(* Logix 5000 project; controller VET 1756-L62 rev 19.52; software revision 19.01; part 4 of 27 *)

        [24].S.BITS1.4   // 7-RED-1024 Cmd. Automatico
        [24].S.BITS1.29   // 90-CAN-011 Falla Abrir
        [24].S.BITS2.20   // 7-RED-1024 Reset Falla
        [24].S.BITS2.23   // 7-RED-1024 Test
        [24].S.BITS2.31   // 90-CAN-011 OUT OPEN
        [28].S.BITS1.0   // 90-VEN-006 Enable
        [28].S.BITS1.1   // 90-VEN-006 Falla Resumen
        [28].S.BITS1.2   // 90-VEN-006 Conf. Marcha
        [28].S.BITS1.4   // 90-VEN-006 Cmd. Automatico
        [28].S.BITS1.26   // 90-VEN-006 FLL
        [28].S.BITS1.27   // 90-VEN-006 FV0
        [28].S.BITS1.28   // 90-VEN-006 FATO
        [28].S.BITS1.30   // 90-VEN-006 Falla Partida
        [28].S.BITS2.27   // 90-VEN-006 Cmd. Marcha
        [28].S.BITS2.20   // 90-VEN-006 Reset Falla
        [28].S.BITS2.23   // 90-VEN-006 Test
        [28].S.BITS2.30   // 90-VEN-006 OUT MARCHA
        [29].S.BITS1.0   // 7-RED-1050 Enable
        [29].S.BITS1.1   // 7-RED-1050 Falla Resumen
        [29].S.BITS1.2   // 7-RED-1050 Conf. Marcha
        [29].S.BITS1.4   // 7-RED-1050 Cmd. Automatico
        [29].S.BITS1.26   // 7-RED-1050 FLL
        [29].S.BITS1.27   // 7-RED-1050 FV0
        [29].S.BITS1.28   // 7-RED-1050 FATO
        [29].S.BITS1.30   // 7-RED-1050 Falla Partida
        [29].S.BITS2.27   // 7-RED-1050 Cmd. Marcha
        [29].S.BITS2.20   // 7-RED-1050 Reset Falla
        [29].S.BITS2.23   // 7-RED-1050 Test
        [29].S.BITS2.30   // 7-RED-1050 OUT MARCHA
        [31].S.BITS1.8   // 90-TOL-001 LL
        [31].S.BITS1.9   // 90-TOL-001 LM
        [31].S.BITS1.10   // 90-TOL-001 LH
        [33].S.BITS1.10   // 90-TOL-003 LH
        [33].S.BITS1.8   // 90-TOL-003 LL
        [33].S.BITS1.9   // 90-TOL-003 LM
        [35].S.BITS1.8   // 90-TOL-005 LL
        [34].S.BITS1.8   // 90-TOL-004 LL
        [37].S.BITS1.10   // 90-TOL-007 LH
        [36].S.BITS1.8   // 7-BIN-1060 LL
        [37].S.BITS1.8   // 90-TOL-007 LL
        [37].S.BITS1.9   // 90-TOL-007 LM
        [40].S.BITS2.30   // 7-VRT-1064 OUT MARCHA
        [43].S.BITS2.30   // 7-VEN-1067 OUT MARCHA
        [44].S.BITS1.2   // 90-FIL-001 Conf Pos Abrir
        [44].S.BITS1.29   // 90-FIL-001 Falla Abrir
        [44].S.BITS2.31   // 90-FIL-001 OUT OPEN
        [45].S.BITS1.26   // 7-ROS-1068 FLL
        [45].S.BITS1.27   // 7-ROS-1068 FV0
        [45].S.BITS1.28   // 7-ROS-1068 FATO
        [45].S.BITS1.30   // 7-ROS-1068 Falla Partida
        [45].S.BITS2.27   // 7-ROS-1068 Cmd. Marcha
        [45].S.BITS2.30   // 7-ROS-1068 OUT MARCHA
        [47].S.BITS1.8   // TV-1 LL
        [47].S.BITS1.10   // TV-1 LH
        [55].S.BITS1.2   // 7-RED-1078 Conf. Marcha
        [55].S.BITS1.29   // 90-FIL-002 Falla Abrir
        [55].S.BITS2.31   // 90-FIL-002 OUT OPEN
        [56].S.BITS1.26   // 90-VEN-002 FLL
        [56].S.BITS1.27   // 90-VEN-002 FV0
        [56].S.BITS1.28   // 90-VEN-002 FATO
        [56].S.BITS1.30   // 7-CON-1079 Falla Cerrar
        [56].S.BITS2.27   // 7-CON-1079 Cmd. Open
        [56].S.BITS2.30   // 7-CON-1079 OUT CLOSE
        [59].S.BITS1.27   // 90-TOR-002 FV0
        [58].S.BITS1.8   // TV-2 LL
        [59].S.BITS1.0   // 90-TOR-002 Enable
        [59].S.BITS1.1   // 90-TOR-002 Falla Resumen
        [59].S.BITS1.2   // 90-TOR-002 Conf. Marcha
        [59].S.BITS1.4   // 90-TOR-002 Cmd. Automatico
        [59].S.BITS1.26   // 90-TOR-002 FLL
        [59].S.BITS1.28   // 90-TOR-002 FATO
        [59].S.BITS1.30   // 90-TOR-002 Falla Partida
        [59].S.BITS2.27   // 90-TOR-002 Cmd. Marcha
        [59].S.BITS2.20   // 90-TOR-002 Reset Falla
        [59].S.BITS2.23   // 90-TOR-002 Test
        [59].S.BITS2.30   // 90-TOR-002 OUT MARCHA
        [63].S.BITS1.0   // 7-MRO-1083c Enable
        [63].S.BITS1.1   // 7-MRO-1083c Falla Resumen
        [63].S.BITS1.2   // 7-MRO-1083c Conf. Marcha
        [63].S.BITS1.4   // 7-MRO-1083c Cmd. Automatico
        [63].S.BITS1.26   // 7-MRO-1083c FLL
        [63].S.BITS1.27   // 7-MRO-1083c FV0
        [63].S.BITS1.28   // 7-MRO-1083c FATO
        [63].S.BITS1.30   // 7-MRO-1083c Falla Partida
        [63].S.BITS2.27   // 7-MRO-1083c Cmd. Marcha
        [63].S.BITS2.20   // 7-MRO-1083c Reset Falla
        [63].S.BITS2.23   // 7-MRO-1083c Test
        [63].S.BITS2.30   // 7-MRO-1083c OUT MARCHA
        [64].S.BITS1.0   // 7-MRO-1083d Enable
        [64].S.BITS1.1   // 7-MRO-1083d Falla Resumen
        [64].S.BITS1.2   // 7-MRO-1083d Conf. Marcha
        [64].S.BITS1.4   // 7-MRO-1083d Cmd. Automatico
        [64].S.BITS1.26   // 7-MRO-1083d FLL
        [64].S.BITS1.27   // 7-MRO-1083d FV0
        [64].S.BITS1.28   // 7-MRO-1083d FATO
        [64].S.BITS1.30   // 7-MRO-1083d Falla Partida
        [64].S.BITS2.27   // 7-MRO-1083d Cmd. Marcha
        [64].S.BITS2.20   // 7-MRO-1083d Reset Falla
        [64].S.BITS2.23   // 7-MRO-1083d Test
        [64].S.BITS2.30   // 7-MRO-1083d OUT MARCHA
        [65].S.BITS1.0   // 90-MRO-001-C Enable
        [65].S.BITS1.1   // 90-MRO-001-C Falla Resumen
        [65].S.BITS1.2   // 90-MRO-001-C Conf. Marcha
        [65].S.BITS1.4   // 90-MRO-001-C Cmd. Automatico
        [65].S.BITS1.26   // 90-MRO-001-C FLL
        [65].S.BITS1.27   // 90-MRO-001-C FV0
        [65].S.BITS1.28   // 90-MRO-001-C FATO
        [65].S.BITS1.30   // 90-MRO-001-C Falla Partida
        [65].S.BITS2.27   // 90-MRO-001-C Cmd. Marcha
        [65].S.BITS2.20   // 90-MRO-001-C Reset Falla
        [65].S.BITS2.23   // 90-MRO-001-C Test
        [65].S.BITS2.30   // 90-MRO-001-C OUT MARCHA
        [72].S.BITS1.2   // 90-ALI-004 Conf. Marcha
        [73].S.BITS1.0   // 7-MRO-1089a Enable
        [73].S.BITS1.1   // 7-MRO-1089a Falla Resumen
        [73].S.BITS1.2   // 7-MRO-1089a Conf. Marcha
        [73].S.BITS1.4   // 7-MRO-1089a Cmd. Automatico
        [73].S.BITS1.26   // 7-MRO-1089a FLL
        [73].S.BITS1.27   // 7-MRO-1089a FV0
        [73].S.BITS1.28   // 7-MRO-1089a FATO
        [73].S.BITS1.30   // 7-MRO-1089a Falla Partida
        [73].S.BITS2.27   // 7-MRO-1089a Cmd. Marcha
        [73].S.BITS2.20   // 7-MRO-1089a Reset Falla
        [73].S.BITS2.23   // 7-MRO-1089a Test
        [73].S.BITS2.30   // 7-MRO-1089a OUT MARCHA
        [74].S.BITS1.0   // 7-MRO-1089b Enable
        [74].S.BITS1.1   // 7-MRO-1089b Falla Resumen
        [74].S.BITS1.4   // 7-MRO-1089b Cmd. Automatico
        [74].S.BITS1.26   // 7-MRO-1089b FLL
        [74].S.BITS1.27   // 7-MRO-1089b FV0
        [74].S.BITS1.28   // 7-MRO-1089b FATO
        [74].S.BITS1.30   // 7-MRO-1089b Falla Partida
        [74].S.BITS2.27   // 7-MRO-1089b Cmd. Marcha
        [74].S.BITS2.20   // 7-MRO-1089b Reset Falla
        [74].S.BITS2.23   // 7-MRO-1089b Test
        [74].S.BITS2.30   // 7-MRO-1089b OUT MARCHA
        [75].S.BITS1.0   // 7-MRO-1089c Enable
        [75].S.BITS1.1   // 7-MRO-1089c Falla Resumen
        [75].S.BITS1.2   // 7-MRO-1089c Conf. Marcha
        [75].S.BITS1.4   // 7-MRO-1089c Cmd. Automatico
        [75].S.BITS1.26   // 7-MRO-1089c FLL
        [75].S.BITS1.27   // 7-MRO-1089c FV0
        [75].S.BITS1.28   // 7-MRO-1089c FATO
        [75].S.BITS1.30   // 7-MRO-1089c Falla Partida
        [75].S.BITS2.27   // 7-MRO-1089c Cmd. Marcha
        [75].S.BITS2.20   // 7-MRO-1089c Reset Falla
        [75].S.BITS2.23   // 7-MRO-1089c Test
        [75].S.BITS2.30   // 7-MRO-1089c OUT MARCHA
        [82].S.BITS1.0   // 7-CON-1095 Enable
        [82].S.BITS1.1   // 7-CON-1095 Falla Resumen
        [82].S.BITS1.4   // 7-CON-1095 Conf Pos Cerrar
        [82].S.BITS1.26   // 90-ALI-005 FLL
        [82].S.BITS1.27   // 90-ALI-005 FV0
        [82].S.BITS1.28   // 90-ALI-005 FATO
        [82].S.BITS1.30   // 7-CON-1095 Falla Cerrar
        [82].S.BITS2.27   // 7-CON-1095 Cmd. Open
        [82].S.BITS2.20   // 7-CON-1095 Reset Falla
        [82].S.BITS2.23   // 7-CON-1095 Test
        [82].S.BITS2.30   // 7-CON-1095 OUT CLOSE
        [83].S.BITS1.0   // 7-CON-1096 Enable
        [83].S.BITS1.1   // 7-CON-1096 Falla Resumen
        [83].S.BITS1.2   // 7-CON-1096 Conf Pos Abrir
        [83].S.BITS1.4   // 7-CON-1096 Conf Pos Cerrar
        [83].S.BITS1.26   // 90-MRO-003-A FLL
        [83].S.BITS1.27   // 90-MRO-003-A FV0
        [83].S.BITS1.28   // 90-MRO-003-A FATO
        [83].S.BITS1.30   // 7-CON-1096 Falla Cerrar
        [83].S.BITS2.27   // 7-CON-1096 Cmd. Open
        [83].S.BITS2.20   // 7-CON-1096 Reset Falla
        [83].S.BITS2.23   // 7-CON-1096 Test
        [83].S.BITS2.30   // 7-CON-1096 OUT CLOSE
        [84].S.BITS1.0   // 7-CON-1097 Enable
        [84].S.BITS1.1   // 7-CON-1097 Falla Resumen
        [84].S.BITS1.4   // 7-CON-1097 Conf Pos Cerrar
        [84].S.BITS1.26   // 90-MRO-003-B FLL
        [84].S.BITS1.27   // 90-MRO-003-B FV0
        [84].S.BITS1.28   // 90-MRO-003-B FATO
        [84].S.BITS1.30   // 7-CON-1097 Falla Cerrar
        [84].S.BITS2.27   // 7-CON-1097 Cmd. Open
        [84].S.BITS2.20   // 7-CON-1097 Reset Falla
        [84].S.BITS2.23   // 7-CON-1097 Test
        [84].S.BITS2.30   // 7-CON-1097 OUT CLOSE
        [85].S.BITS1.0   // 90-MRO-003-C Enable
        [85].S.BITS1.1   // 90-MRO-003-C Falla Resumen
        [85].S.BITS1.4   // 90-MRO-003-C Cmd. Automatico
        [85].S.BITS1.26   // 90-MRO-003-C FLL
        [85].S.BITS1.27   // 90-MRO-003-C FV0
        [85].S.BITS1.28   // 90-MRO-003-C FATO
        [85].S.BITS1.30   // 90-MRO-003-C Falla Partida
        [85].S.BITS2.27   // 90-MRO-003-C Cmd. Marcha
        [85].S.BITS2.20   // 90-MRO-003-C Reset Falla
        [85].S.BITS2.23   // 90-MRO-003-C Test
        [85].S.BITS2.30   // 90-MRO-003-C OUT MARCHA
        [92].S.BITS1.0   // 90-VEN-003 Enable
        [92].S.BITS1.1   // 90-VEN-003 Falla Resumen
        [92].S.BITS1.2   // 90-VEN-003 Conf. Marcha
        [92].S.BITS1.4   // 90-VEN-003 Cmd. Automatico
        [92].S.BITS1.26   // 90-VEN-003 FLL
        [92].S.BITS1.27   // 90-VEN-003 FV0
        [92].S.BITS1.28   // 90-VEN-003 FATO
        [92].S.BITS1.30   // 90-VEN-003 Falla Partida
        [92].S.BITS2.27   // 90-VEN-003 Cmd. Marcha
        [92].S.BITS2.20   // 90-VEN-003 Reset Falla
        [92].S.BITS2.23   // 90-VEN-003 Test
        [92].S.BITS2.30   // 90-VEN-003 OUT MARCHA
        [96].S.BITS1.27   // 90-TDC-006 FV0
        [94].S.BITS1.8   // 90-TOL-008 LL
        [94].S.BITS1.9   // 90-TOL-008 LM
        [94].S.BITS1.10   // 90-TOL-008 LH
        [96].S.BITS1.0   // 90-TDC-006 Enable
        [96].S.BITS1.1   // 90-TDC-006 Falla Resumen
        [96].S.BITS1.4   // 90-TDC-006 Cmd. Automatico
        [96].S.BITS1.26   // 90-TDC-006 FLL
        [96].S.BITS1.28   // 90-TDC-006 FATO
        [96].S.BITS1.30   // 90-TDC-006 Falla Partida
        [96].S.BITS2.27   // 90-TDC-006 Cmd. Marcha
        [96].S.BITS2.20   // 90-TDC-006 Reset Falla
        [96].S.BITS2.23   // 90-TDC-006 Test
        [96].S.BITS2.30   // 90-TDC-006 OUT MARCHA
        [97].S.BITS1.0   // 90-CAN-019 Enable
        [97].S.BITS1.1   // 90-CAN-019 Falla Resumen
        [97].S.BITS1.2   // 90-CAN-019 Conf Pos Abrir
        [97].S.BITS1.4   // 90-CAN-019 Conf Pos Cerrar
        [97].S.BITS1.29   // 90-CAN-019 Falla Abrir
        [97].S.BITS1.30   // 90-CAN-019 Falla Cerrar
        [97].S.BITS2.20   // 90-CAN-019 Reset Falla
        [97].S.BITS2.23   // 90-CAN-019 Test
        [97].S.BITS2.27   // 90-CAN-019 Cmd. Open
        [97].S.BITS2.30   // 90-CAN-019 OUT CLOSE
        [97].S.BITS2.31   // 90-CAN-019 OUT OPEN
        [101].S.BITS1.8   // 7-BIN-1100 LL
        [99].S.BITS1.9   // TOLVIR-MRO1 LM
        [102].S.BITS1.1   // 7-ROS-1101 Falla Resumen
        [100].S.BITS1.8   // TOLVIR-MRO2 LL
        [100].S.BITS1.9   // TOLVIR-MRO2 LM
        [100].S.BITS1.10   // TOLVIR-MRO2 LH
        [102].S.BITS1.27   // 7-ROS-1101 FV0
        [101].S.BITS1.9   // 7-BIN-1100 LM
        [101].S.BITS1.10   // 7-BIN-1100 LH
        [102].S.BITS1.0   // 7-ROS-1101 Enable
        [102].S.BITS1.2   // 7-ROS-1101 Conf. Marcha
        [102].S.BITS1.4   // 7-ROS-1101 Cmd. Automatico
        [102].S.BITS1.26   // 7-ROS-1101 FLL
        [102].S.BITS1.28   // 7-ROS-1101 FATO
        [102].S.BITS1.30   // 7-ROS-1101 Falla Partida
        [102].S.BITS2.27   // 7-ROS-1101 Cmd. Marcha
        [102].S.BITS2.20   // 7-ROS-1101 Reset Falla
        [102].S.BITS2.23   // 7-ROS-1101 Test
        [102].S.BITS2.30   // 7-ROS-1101 OUT MARCHA
        [104].S.BITS1.0   // 7-ROS-1103 Enable
        [104].S.BITS1.1   // 7-ROS-1103 Falla Resumen
        [104].S.BITS1.2   // 7-ROS-1103 Conf. Marcha
        [104].S.BITS1.4   // 7-ROS-1103 Cmd. Automatico
        [104].S.BITS1.26   // 7-ROS-1103 FLL
        [104].S.BITS1.27   // 7-ROS-1103 FV0
        [104].S.BITS1.28   // 7-ROS-1103 FATO
        [104].S.BITS1.30   // 7-ROS-1103 Falla Partida
        [104].S.BITS2.27   // 7-ROS-1103 Cmd. Marcha
        [104].S.BITS2.20   // 7-ROS-1103 Reset Falla
        [104].S.BITS2.23   // 7-ROS-1103 Test
        [104].S.BITS2.30   // 7-ROS-1103 OUT MARCHA
        [105].S.BITS1.0   // 90-TDC-004 Enable
        [105].S.BITS1.1   // 90-TDC-004 Falla Resumen
        [105].S.BITS1.2   // 90-TDC-004 Conf. Marcha
        [105].S.BITS1.4   // 90-TDC-004 Cmd. Automatico
        [105].S.BITS1.26   // 90-TDC-004 FLL
        [105].S.BITS1.27   // 90-TDC-004 FV0
        [105].S.BITS1.28   // 90-TDC-004 FATO
        [105].S.BITS1.30   // 90-TDC-004 Falla Partida
        [105].S.BITS2.27   // 90-TDC-004 Cmd. Marcha
        [105].S.BITS2.20   // 90-TDC-004 Reset Falla
        [105].S.BITS2.23   // 90-TDC-004 Test
        [105].S.BITS2.30   // 90-TDC-004 OUT MARCHA
        [106].S.BITS1.0   // 7-ROS-1105 Enable
        [106].S.BITS1.1   // 7-ROS-1105 Falla Resumen
        [106].S.BITS1.4   // 7-ROS-1105 Cmd. Automatico
        [106].S.BITS1.26   // 7-ROS-1105 FLL
        [106].S.BITS1.27   // 7-ROS-1105 FV0
        [106].S.BITS1.28   // 7-ROS-1105 FATO
        [106].S.BITS1.30   // 7-ROS-1105 Falla Partida
        [106].S.BITS2.27   // 7-ROS-1105 Cmd. Marcha
        [106].S.BITS2.20   // 7-ROS-1105 Reset Falla
        [106].S.BITS2.23   // 7-ROS-1105 Test
        [106].S.BITS2.30   // 7-ROS-1105 OUT MARCHA
        [107].S.BITS1.0   // 90-ELV-002 Enable
        [107].S.BITS1.1   // 90-ELV-002 Falla Resumen
        [107].S.BITS1.2   // 90-ELV-002 Conf. Marcha
        [107].S.BITS1.4   // 90-ELV-002 Cmd. Automatico
        [107].S.BITS1.26   // 90-ELV-002 FLL
        [107].S.BITS1.27   // 90-ELV-002 FV0
        [107].S.BITS1.28   // 90-ELV-002 FATO
        [107].S.BITS1.30   // 90-ELV-002 Falla Partida
        [107].S.BITS2.27   // 90-ELV-002 Cmd. Marcha
        [107].S.BITS2.20   // 90-ELV-002 Reset Falla
        [107].S.BITS2.23   // 90-ELV-002 Test
        [107].S.BITS2.30   // 90-ELV-002 OUT MARCHA
        [109].S.BITS1.0   // 90-ELV-004 Enable
        [109].S.BITS1.1   // 90-ELV-004 Falla Resumen
        [109].S.BITS1.4   // 90-ELV-004 Cmd. Automatico
        [109].S.BITS1.26   // 90-ELV-004 FLL
        [109].S.BITS1.27   // 90-ELV-004 FV0
        [109].S.BITS1.28   // 90-ELV-004 FATO
        [109].S.BITS1.30   // 90-ELV-004 Falla Partida
        [109].S.BITS2.27   // 90-ELV-004 Cmd. Marcha
        [109].S.BITS2.20   // 90-ELV-004 Reset Falla
        [109].S.BITS2.23   // 90-ELV-004 Test
        [109].S.BITS2.30   // 90-ELV-004 OUT MARCHA
        [112].S.BITS1.0   // 7-ROS-1111 Enable
        [112].S.BITS1.1   // 7-ROS-1111 Falla Resumen
        [112].S.BITS1.2   // 7-ROS-1111 Conf. Marcha
        [112].S.BITS1.4   // 7-ROS-1111 Cmd. Automatico
        [112].S.BITS1.26   // 7-ROS-1111 FLL
        [112].S.BITS1.27   // 7-ROS-1111 FV0
        [112].S.BITS1.28   // 7-ROS-1111 FATO
        [112].S.BITS1.30   // 7-ROS-1111 Falla Partida
        [112].S.BITS2.27   // 7-ROS-1111 Cmd. Marcha
        [112].S.BITS2.20   // 7-ROS-1111 Reset Falla
        [112].S.BITS2.23   // 7-ROS-1111 Test
        [112].S.BITS2.30   // 7-ROS-1111 OUT MARCHA
        [113].S.BITS1.0   // 100-VEN-001 Enable
        [113].S.BITS1.1   // 100-VEN-001 Falla Resumen
        [113].S.BITS1.2   // 100-VEN-001 Conf. Marcha
        [113].S.BITS1.4   // 100-VEN-001 Cmd. Automatico
        [113].S.BITS1.26   // 100-VEN-001 FLL
        [113].S.BITS1.27   // 100-VEN-001 FV0
        [113].S.BITS1.28   // 100-VEN-001 FATO
        [113].S.BITS1.30   // 100-VEN-001 Falla Partida
        [113].S.BITS2.27   // 100-VEN-001 Cmd. Marcha
        [113].S.BITS2.20   // 100-VEN-001 Reset Falla
        [113].S.BITS2.23   // 100-VEN-001 Test
        [113].S.BITS2.30   // 100-VEN-001 OUT MARCHA
        [115].S.BITS1.27   // 100-TOR-022 FV0
        [114].S.BITS1.8   // 100-TOL-005 LL
        [114].S.BITS1.9   // 100-TOL-005 LM
        [114].S.BITS1.10   // 100-TOL-005 LH
        [115].S.BITS1.0   // 100-TOR-022 Enable
        [115].S.BITS1.1   // 100-TOR-022 Falla Resumen
        [115].S.BITS1.4   // 100-TOR-022 Cmd. Automatico
        [115].S.BITS1.26   // 100-TOR-022 FLL
        [115].S.BITS1.28   // 100-TOR-022 FATO
        [115].S.BITS1.30   // 100-TOR-022 Falla Partida
        [115].S.BITS2.27   // 100-TOR-022 Cmd. Marcha
        [115].S.BITS2.20   // 100-TOR-022 Reset Falla
        [115].S.BITS2.23   // 100-TOR-022 Test
        [115].S.BITS2.30   // 100-TOR-022 OUT MARCHA
        [116].S.BITS1.0   // 7-ROS-1115 Enable
        [116].S.BITS1.1   // 7-ROS-1115 Falla Resumen
        [116].S.BITS1.4   // 7-ROS-1115 Cmd. Automatico
        [116].S.BITS1.26   // 7-ROS-1115 FLL
        [116].S.BITS1.27   // 7-ROS-1115 FV0
        [116].S.BITS1.28   // 7-ROS-1115 FATO
        [116].S.BITS1.30   // 7-ROS-1115 Falla Partida
        [116].S.BITS2.27   // 7-ROS-1115 Cmd. Marcha
        [116].S.BITS2.20   // 7-ROS-1115 Reset Falla
        [116].S.BITS2.23   // 7-ROS-1115 Test
        [116].S.BITS2.30   // 7-ROS-1115 OUT MARCHA
        [117].S.BITS1.0   // 100-BIF-001 Enable
        [117].S.BITS1.1   // 100-BIF-001 Falla Resumen
        [117].S.BITS1.2   // 100-BIF-001 Conf. Pos. Izquierda
        [117].S.BITS1.4   // 100-BIF-001 Conf. Pos. Derecha
        [117].S.BITS1.29   // 100-BIF-001 Falla Pos. Izquierda
        [117].S.BITS1.30   // 100-BIF-001 Falla Pos. Derecha
        [117].S.BITS2.20   // 100-BIF-001 Reset Falla
        [117].S.BITS2.23   // 100-BIF-001 Test
        [117].S.BITS2.26   // 100-BIF-001 Cmd. Pos . Izquierda
        [117].S.BITS2.27   // 100-BIF-001 Cmd. Pos. Derecha
        [117].S.BITS2.30   // 100-BIF-001 Out Izquierda
        [117].S.BITS2.31   // 100-BIF-001 Out Derecha
        [122].S.BITS1.0   // 7-ROS-1121 Enable
        [122].S.BITS1.1   // 7-ROS-1121 Falla Resumen
        [122].S.BITS1.2   // 7-ROS-1121 Conf. Marcha
        [122].S.BITS1.4   // 7-ROS-1121 Cmd. Automatico
        [122].S.BITS1.26   // 7-ROS-1121 FLL
        [122].S.BITS1.27   // 7-ROS-1121 FV0
        [122].S.BITS1.28   // 7-ROS-1121 FATO
        [122].S.BITS1.30   // 7-ROS-1121 Falla Partida
        [122].S.BITS2.27   // 7-ROS-1121 Cmd. Marcha
        [122].S.BITS2.20   // 7-ROS-1121 Reset Falla
        [122].S.BITS2.23   // 7-ROS-1121 Test
        [122].S.BITS2.30   // 7-ROS-1121 OUT MARCHA
        [123].S.BITS1.0   // 100-CAN-018 Enable
        [123].S.BITS1.1   // 100-CAN-018 Falla Resumen
        [123].S.BITS1.2   // 100-CAN-018 Conf Pos Abrir
        [123].S.BITS1.4   // 100-CAN-018 Conf Pos Cerrar
        [123].S.BITS1.29   // 100-CAN-018 Falla Abrir
        [123].S.BITS2.20   // 100-CAN-018 Reset Falla
        [123].S.BITS2.23   // 100-CAN-018 Test
        [123].S.BITS2.31   // 100-CAN-018 OUT OPEN
        [124].S.BITS1.0   // 7-ROS-1123 Enable
        [124].S.BITS1.1   // 7-ROS-1123 Falla Resumen
        [124].S.BITS1.2   // 7-ROS-1123 Conf. Marcha
        [124].S.BITS1.4   // 7-ROS-1123 Cmd. Automatico
        [124].S.BITS1.29   // 100-CAN-019 Falla Abrir
        [124].S.BITS1.30   // 7-ROS-1123 Falla Partida
        [124].S.BITS2.20   // 7-ROS-1123 Reset Falla
        [124].S.BITS2.23   // 7-ROS-1123 Test
        [124].S.BITS2.30   // 7-ROS-1123 OUT MARCHA
        [124].S.BITS2.31   // 100-CAN-019 OUT OPEN
        [126].S.BITS1.0   // 7-ROS-1125 Enable
        [126].S.BITS1.1   // 7-ROS-1125 Falla Resumen
        [126].S.BITS1.2   // 7-ROS-1125 Conf. Marcha
        [126].S.BITS1.4   // 7-ROS-1125 Cmd. Automatico
        [126].S.BITS1.26   // 7-ROS-1125 FLL
        [126].S.BITS1.27   // 7-ROS-1125 FV0
        [126].S.BITS1.28   // 7-ROS-1125 FATO
        [126].S.BITS1.30   // 7-ROS-1125 Falla Partida
        [126].S.BITS2.27   // 7-ROS-1125 Cmd. Marcha
        [126].S.BITS2.20   // 7-ROS-1125 Reset Falla
        [126].S.BITS2.23   // 7-ROS-1125 Test
        [126].S.BITS2.30   // 7-ROS-1125 OUT MARCHA
        [127].S.BITS1.0   // 100-CAN-020 Enable
        [127].S.BITS1.1   // 100-CAN-020 Falla Resumen
        [127].S.BITS1.2   // 100-CAN-020 Conf Pos Abrir
        [127].S.BITS1.4   // 100-CAN-020 Conf Pos Cerrar
        [127].S.BITS1.29   // 100-CAN-020 Falla Abrir
        [127].S.BITS2.20   // 100-CAN-020 Reset Falla
        [127].S.BITS2.23   // 100-CAN-020 Test
        [127].S.BITS2.31   // 100-CAN-020 OUT OPEN
        [128].S.BITS1.0   // 7-ROS-1127 Enable
        [128].S.BITS1.1   // 7-ROS-1127 Falla Resumen
        [128].S.BITS1.2   // 7-ROS-1127 Conf. Marcha
        [128].S.BITS1.4   // 7-ROS-1127 Cmd. Automatico
        [128].S.BITS1.29   // 100-CAN-021 Falla Abrir
        [128].S.BITS1.30   // 7-ROS-1127 Falla Partida
        [128].S.BITS2.20   // 7-ROS-1127 Reset Falla
        [128].S.BITS2.23   // 7-ROS-1127 Test
        [128].S.BITS2.30   // 7-ROS-1127 OUT MARCHA
        [128].S.BITS2.31   // 100-CAN-021 OUT OPEN
        [131].S.BITS1.0   // 100-TDC-001 Enable
        [131].S.BITS1.1   // 100-TDC-001 Falla Resumen
        [131].S.BITS1.4   // 100-TDC-001 Cmd. Automatico
        [131].S.BITS1.26   // 100-TDC-001 FLL
        [131].S.BITS1.27   // 100-TDC-001 FV0
        [131].S.BITS1.28   // 100-TDC-001 FATO
        [131].S.BITS1.30   // 100-TDC-001 Falla Partida
        [131].S.BITS2.27   // 100-TDC-001 Cmd. Marcha
        [131].S.BITS2.20   // 100-TDC-001 Reset Falla
        [131].S.BITS2.23   // 100-TDC-001 Test
        [131].S.BITS2.30   // 100-TDC-001 OUT MARCHA
        [132].S.BITS1.0   // 100-CAN-001 Enable
        [132].S.BITS1.1   // 100-CAN-001 Falla Resumen
        [132].S.BITS1.2   // 100-CAN-001 Conf Pos Abrir
        [132].S.BITS1.4   // 100-CAN-001 Conf Pos Cerrar
        [132].S.BITS1.29   // 100-CAN-001 Falla Abrir
        [132].S.BITS1.30   // 100-CAN-001 Falla Cerrar
        [132].S.BITS2.20   // 100-CAN-001 Reset Falla
        [132].S.BITS2.23   // 100-CAN-001 Test
        [132].S.BITS2.27   // 100-CAN-001 Cmd. Open
        [132].S.BITS2.30   // 100-CAN-001 OUT CLOSE
        [132].S.BITS2.31   // 100-CAN-001 OUT OPEN
        [134].S.BITS1.0   // 100-TDC-002 Enable
        [134].S.BITS1.1   // 100-TDC-002 Falla Resumen
        [134].S.BITS1.2   // 100-TDC-002 Conf. Marcha
        [134].S.BITS1.4   // 100-TDC-002 Cmd. Automatico
        [134].S.BITS1.26   // 100-TDC-002 FLL
        [134].S.BITS1.27   // 100-TDC-002 FV0
        [134].S.BITS1.28   // 100-TDC-002 FATO
        [134].S.BITS1.30   // 100-TDC-002 Falla Partida
        [134].S.BITS2.27   // 100-TDC-002 Cmd. Marcha
        [134].S.BITS2.20   // 100-TDC-002 Reset Falla
        [134].S.BITS2.23   // 100-TDC-002 Test
        [134].S.BITS2.30   // 100-TDC-002 OUT MARCHA
        [135].S.BITS1.0   // 100-CAN-002 Enable
        [135].S.BITS1.1   // 100-CAN-002 Falla Resumen
        [135].S.BITS1.2   // 100-CAN-002 Conf Pos Abrir
        [135].S.BITS1.4   // 100-CAN-002 Conf Pos Cerrar
        [135].S.BITS1.29   // 100-CAN-002 Falla Abrir
        [135].S.BITS1.30   // 100-CAN-002 Falla Cerrar
        [135].S.BITS2.20   // 100-CAN-002 Reset Falla
        [135].S.BITS2.23   // 100-CAN-002 Test
        [135].S.BITS2.27   // 100-CAN-002 Cmd. Open
        [135].S.BITS2.30   // 100-CAN-002 OUT CLOSE
        [135].S.BITS2.31   // 100-CAN-002 OUT OPEN
        [136].S.BITS1.0   // 100-CAN-003 Enable
        [136].S.BITS1.1   // 100-CAN-003 Falla Resumen
        [136].S.BITS1.2   // 100-CAN-003 Conf Pos Abrir
        [136].S.BITS1.4   // 100-CAN-003 Conf Pos Cerrar
        [136].S.BITS1.29   // 100-CAN-003 Falla Abrir
        [136].S.BITS1.30   // 100-CAN-003 Falla Cerrar
        [136].S.BITS2.20   // 100-CAN-003 Reset Falla
        [136].S.BITS2.23   // 100-CAN-003 Test
        [136].S.BITS2.27   // 100-CAN-003 Cmd. Open
        [136].S.BITS2.30   // 100-CAN-003 OUT CLOSE
        [137].S.BITS1.0   // 100-CAN-004 Enable
        [137].S.BITS1.1   // 100-CAN-004 Falla Resumen
        [137].S.BITS1.2   // 100-CAN-004 Conf Pos Abrir
        [137].S.BITS1.4   // 100-CAN-004 Conf Pos Cerrar
        [137].S.BITS1.29   // 100-CAN-004 Falla Abrir
        [137].S.BITS1.30   // 100-CAN-004 Falla Cerrar
        [137].S.BITS2.20   // 100-CAN-004 Reset Falla
        [137].S.BITS2.23   // 100-CAN-004 Test
        [137].S.BITS2.27   // 100-CAN-004 Cmd. Open
        [137].S.BITS2.30   // 100-CAN-004 OUT CLOSE
        [137].S.BITS2.31   // 100-CAN-004 OUT OPEN
        [142].S.BITS1.0   // 7-FIL-1141 Enable
        [142].S.BITS1.1   // 7-FIL-1141 Falla Resumen
        [142].S.BITS1.2   // 7-FIL-1141 Conf. Marcha
        [142].S.BITS1.4   // 7-FIL-1141 Cmd. Automatico
        [142].S.BITS1.26   // 7-FIL-1141 FLL
        [142].S.BITS1.27   // 7-FIL-1141 FV0
        [142].S.BITS1.28   // 7-FIL-1141 FATO
        [142].S.BITS1.30   // 7-FIL-1141 Falla Partida
        [142].S.BITS2.27   // 7-FIL-1141 Cmd. Marcha
        [142].S.BITS2.20   // 7-FIL-1141 Reset Falla
        [142].S.BITS2.23   // 7-FIL-1141 Test
        [142].S.BITS2.30   // 7-FIL-1141 OUT MARCHA
        [143].S.BITS1.0   // 7-BBA-1142 Enable
        [143].S.BITS1.1   // 7-BBA-1142 Falla Resumen
        [143].S.BITS1.2   // 7-BBA-1142 Conf. Marcha
        [143].S.BITS1.4   // 7-BBA-1142 Cmd. Automatico
        [143].S.BITS1.29   // 100-CAN-005 Falla Abrir
        [143].S.BITS2.20   // 7-BBA-1142 Reset Falla
        [143].S.BITS2.23   // 7-BBA-1142 Test
        [143].S.BITS2.31   // 100-CAN-005 OUT OPEN
        [144].S.BITS1.0   // 7-RED-1143 Enable
        [144].S.BITS1.1   // 7-RED-1143 Falla Resumen
        [144].S.BITS1.2   // 7-RED-1143 Conf. Marcha
        [144].S.BITS1.4   // 7-RED-1143 Cmd. Automatico
        [144].S.BITS1.29   // 100-CAN-006 Falla Abrir
        [144].S.BITS1.30   // 7-RED-1143 Falla Partida
        [144].S.BITS2.20   // 7-RED-1143 Reset Falla
        [144].S.BITS2.23   // 7-RED-1143 Test
        [144].S.BITS2.30   // 7-RED-1143 OUT MARCHA
        [144].S.BITS2.31   // 100-CAN-006 OUT OPEN
        [146].S.BITS1.0   // 7-RED-1145 Enable
        [146].S.BITS1.1   // 7-RED-1145 Falla Resumen
        [146].S.BITS1.2   // 7-RED-1145 Conf. Marcha
        [146].S.BITS1.4   // 7-RED-1145 Cmd. Automatico
        [146].S.BITS1.26   // 7-RED-1145 FLL
        [146].S.BITS1.27   // 7-RED-1145 FV0
        [146].S.BITS1.28   // 7-RED-1145 FATO
        [146].S.BITS1.30   // 7-RED-1145 Falla Partida
        [146].S.BITS2.27   // 7-RED-1145 Cmd. Marcha
        [146].S.BITS2.20   // 7-RED-1145 Reset Falla
        [146].S.BITS2.23   // 7-RED-1145 Test
        [146].S.BITS2.30   // 7-RED-1145 OUT MARCHA
        [147].S.BITS1.0   // 7-CON-1146 Enable
        [147].S.BITS1.1   // 7-CON-1146 Falla Resumen
        [147].S.BITS1.2   // 7-CON-1146 Conf Pos Abrir
        [147].S.BITS1.4   // 7-CON-1146 Conf Pos Cerrar
        [147].S.BITS1.29   // 7-CON-1146 Falla Abrir
        [147].S.BITS2.20   // 7-CON-1146 Reset Falla
        [147].S.BITS2.23   // 7-CON-1146 Test
        [147].S.BITS2.31   // 7-CON-1146 OUT OPEN
        [148].S.BITS1.0   // 7-CON-1147 Enable
        [148].S.BITS1.1   // 7-CON-1147 Falla Resumen
        [148].S.BITS1.2   // 7-CON-1147 Conf Pos Abrir
        [148].S.BITS1.4   // 7-CON-1147 Conf Pos Cerrar
        [148].S.BITS1.29   // 7-CON-1147 Falla Abrir
        [148].S.BITS1.30   // 7-CON-1147 Falla Cerrar
        [148].S.BITS2.20   // 7-CON-1147 Reset Falla
        [148].S.BITS2.23   // 7-CON-1147 Test
        [148].S.BITS2.27   // 7-CON-1147 Cmd. Open
        [148].S.BITS2.30   // 7-CON-1147 OUT CLOSE
        [148].S.BITS2.31   // 7-CON-1147 OUT OPEN
        [152].S.BITS1.0   // 7-CON-1152 Enable
        [152].S.BITS1.1   // 7-CON-1152 Falla Resumen
        [152].S.BITS1.4   // 7-CON-1152 Conf Pos Cerrar
        [152].S.BITS1.26   // 100-TDC-005 FLL
        [152].S.BITS1.27   // 100-TDC-005 FV0
        [152].S.BITS1.28   // 100-TDC-005 FATO
        [152].S.BITS1.30   // 7-CON-1152 Falla Cerrar
        [152].S.BITS2.27   // 7-CON-1152 Cmd. Open
        [152].S.BITS2.20   // 7-CON-1152 Reset Falla
        [152].S.BITS2.23   // 7-CON-1152 Test
        [152].S.BITS2.30   // 7-CON-1152 OUT CLOSE
        [153].S.BITS1.0   // 7-CON-1153 Enable
        [153].S.BITS1.1   // 7-CON-1153 Falla Resumen
        [153].S.BITS1.2   // 7-CON-1153 Conf Pos Abrir
        [153].S.BITS1.4   // 7-CON-1153 Conf Pos Cerrar
        [153].S.BITS1.29   // 7-CON-1153 Falla Abrir
        [153].S.BITS2.20   // 7-CON-1153 Reset Falla
        [153].S.BITS2.23   // 7-CON-1153 Test
        [153].S.BITS2.31   // 7-CON-1153 OUT OPEN
        [154].S.BITS1.0   // 7-ELV-1149 Enable
        [154].S.BITS1.1   // 7-ELV-1149 Falla Resumen
        [154].S.BITS1.2   // 7-ELV-1149 Conf. Marcha
        [154].S.BITS1.4   // 7-ELV-1149 Cmd. Automatico
        [154].S.BITS1.29   // 100-CAN-014 Falla Abrir
        [154].S.BITS1.30   // 7-ELV-1149 Falla Partida
        [154].S.BITS2.20   // 7-ELV-1149 Reset Falla
        [154].S.BITS2.23   // 7-ELV-1149 Test
        [154].S.BITS2.30   // 7-ELV-1149 OUT MARCHA
        [154].S.BITS2.31   // 100-CAN-014 OUT OPEN
        [155].S.BITS1.0   // 100-CAN-015 Enable
        [155].S.BITS1.1   // 100-CAN-015 Falla Resumen
        [155].S.BITS1.2   // 100-CAN-015 Conf Pos Abrir
        [155].S.BITS1.4   // 100-CAN-015 Conf Pos Cerrar
        [155].S.BITS1.29   // 100-CAN-015 Falla Abrir
        [155].S.BITS2.20   // 100-CAN-015 Reset Falla
        [155].S.BITS2.23   // 100-CAN-015 Test
        [155].S.BITS2.31   // 100-CAN-015 OUT OPEN
        [157].S.BITS1.0   // 7-ROS-1156 Enable
        [157].S.BITS1.1   // 7-ROS-1156 Falla Resumen
        [157].S.BITS1.2   // 7-ROS-1156 Conf. Marcha
        [157].S.BITS1.4   // 7-ROS-1156 Cmd. Automatico
        [157].S.BITS1.26   // 7-ROS-1156 FLL
        [157].S.BITS1.27   // 7-ROS-1156 FV0
        [157].S.BITS1.28   // 7-ROS-1156 FATO
        [157].S.BITS1.30   // 7-ROS-1156 Falla Partida
        [157].S.BITS2.27   // 7-ROS-1156 Cmd. Marcha
        [157].S.BITS2.20   // 7-ROS-1156 Reset Falla
        [157].S.BITS2.23   // 7-ROS-1156 Test
        [157].S.BITS2.30   // 7-ROS-1156 OUT MARCHA
        [158].S.BITS1.0   // 100-CAN-016 Enable
        [158].S.BITS1.1   // 100-CAN-016 Falla Resumen
        [158].S.BITS1.2   // 100-CAN-016 Conf Pos Abrir
        [158].S.BITS1.4   // 100-CAN-016 Conf Pos Cerrar
        [158].S.BITS1.29   // 100-CAN-016 Falla Abrir
        [158].S.BITS1.30   // 100-CAN-016 Falla Cerrar
        [158].S.BITS2.20   // 100-CAN-016 Reset Falla
        [158].S.BITS2.23   // 100-CAN-016 Test
        [158].S.BITS2.27   // 100-CAN-016 Cmd. Open
        [158].S.BITS2.30   // 100-CAN-016 OUT CLOSE
        [158].S.BITS2.31   // 100-CAN-016 OUT OPEN
        [159].S.BITS1.0   // 7-ROS-1158 Enable
        [159].S.BITS1.1   // 7-ROS-1158 Falla Resumen
        [159].S.BITS1.2   // 7-ROS-1158 Conf. Marcha
        [159].S.BITS1.4   // 7-ROS-1158 Cmd. Automatico
        [159].S.BITS1.29   // 100-CAN-017 Falla Abrir
        [159].S.BITS2.20   // 7-ROS-1158 Reset Falla
        [159].S.BITS2.23   // 7-ROS-1158 Test
        [159].S.BITS2.31   // 100-CAN-017 OUT OPEN
        [162].S.BITS1.0   // 100-TDC-008 Enable
        [162].S.BITS1.1   // 100-TDC-008 Falla Resumen
        [162].S.BITS1.2   // 100-TDC-008 Conf. Marcha
        [162].S.BITS1.4   // 100-TDC-008 Cmd. Automatico
        [162].S.BITS1.26   // 100-TDC-008 FLL
        [162].S.BITS1.27   // 100-TDC-008 FV0
        [162].S.BITS1.28   // 100-TDC-008 FATO
        [162].S.BITS1.30   // 100-TDC-008 Falla Partida
        [162].S.BITS2.27   // 100-TDC-008 Cmd. Marcha
        [162].S.BITS2.20   // 100-TDC-008 Reset Falla
        [162].S.BITS2.23   // 100-TDC-008 Test
        [162].S.BITS2.30   // 100-TDC-008 OUT MARCHA
        [163].S.BITS1.0   // 7-ROS-1162 Enable
        [163].S.BITS1.1   // 7-ROS-1162 Falla Resumen
        [163].S.BITS1.2   // 7-ROS-1162 Conf. Marcha
        [163].S.BITS1.4   // 7-ROS-1162 Cmd. Automatico
        [163].S.BITS1.29   // 100-CAN-028 Falla Abrir
        [163].S.BITS2.20   // 7-ROS-1162 Reset Falla
        [163].S.BITS2.23   // 7-ROS-1162 Test
        [163].S.BITS2.31   // 100-CAN-028 OUT OPEN
        [164].S.BITS1.0   // 100-BIF-002 Enable
        [164].S.BITS1.1   // 100-BIF-002 Falla Resumen
        [164].S.BITS1.2   // 100-BIF-002 Conf. Pos. Izquierda
        [164].S.BITS1.4   // 100-BIF-002 Conf. Pos. Derecha
        [164].S.BITS1.29   // 100-BIF-002 Falla Pos. Izquierda
        [164].S.BITS1.30   // 100-BIF-002 Falla Pos. Derecha
        [164].S.BITS2.20   // 100-BIF-002 Reset Falla
        [164].S.BITS2.23   // 100-BIF-002 Test
        [164].S.BITS2.26   // 100-BIF-002 Cmd. Pos . Izquierda
        [164].S.BITS2.27   // 100-BIF-002 Cmd. Pos. Derecha
        [164].S.BITS2.30   // 100-BIF-002 Out Izquierda
        [164].S.BITS2.31   // 100-BIF-002 Out Derecha
        [165].S.BITS1.0   // 7-ROS-1164 Enable
        [165].S.BITS1.1   // 7-ROS-1164 Falla Resumen
        [165].S.BITS1.2   // 7-ROS-1164 Conf. Marcha
        [165].S.BITS1.4   // 7-ROS-1164 Cmd. Automatico
        [165].S.BITS1.29   // 100-BIF-003 Falla Pos. Izquierda
        [165].S.BITS1.30   // 7-ROS-1164 Falla Partida
        [165].S.BITS2.20   // 7-ROS-1164 Reset Falla
        [165].S.BITS2.23   // 7-ROS-1164 Test
        [165].S.BITS2.26   // 100-BIF-003 Cmd. Pos . Izquierda
        [165].S.BITS2.27   // 7-ROS-1164 Cmd. Marcha
        [165].S.BITS2.30   // 7-ROS-1164 OUT MARCHA
        [165].S.BITS2.31   // 100-BIF-003 Out Derecha
        [167].S.BITS1.0   // 7-ROS-1166 Enable
        [167].S.BITS1.1   // 7-ROS-1166 Falla Resumen
        [167].S.BITS1.2   // 7-ROS-1166 Conf. Marcha
        [167].S.BITS1.4   // 7-ROS-1166 Cmd. Automatico
        [167].S.BITS1.26   // 7-ROS-1166 FLL
        [167].S.BITS1.27   // 7-ROS-1166 FV0
        [167].S.BITS1.28   // 7-ROS-1166 FATO
        [167].S.BITS1.30   // 7-ROS-1166 Falla Partida
        [167].S.BITS2.27   // 7-ROS-1166 Cmd. Marcha
        [167].S.BITS2.20   // 7-ROS-1166 Reset Falla
        [167].S.BITS2.23   // 7-ROS-1166 Test
        [167].S.BITS2.30   // 7-ROS-1166 OUT MARCHA
        [168].S.BITS1.0   // 100-FIL-002 Enable
        [168].S.BITS1.1   // 100-FIL-002 Falla Resumen
        [168].S.BITS1.2   // 100-FIL-002 Conf. Marcha
        [168].S.BITS1.4   // 100-FIL-002 Cmd. Automatico
        [168].S.BITS1.26   // 100-FIL-002 FLL
        [168].S.BITS1.27   // 100-FIL-002 FV0
        [168].S.BITS1.28   // 100-FIL-002 FATO
        [168].S.BITS1.30   // 100-FIL-002 Falla Partida
        [168].S.BITS2.27   // 100-FIL-002 Cmd. Marcha
        [168].S.BITS2.20   // 100-FIL-002 Reset Falla
        [168].S.BITS2.23   // 100-FIL-002 Test
        [168].S.BITS2.30   // 100-FIL-002 OUT MARCHA
        [169].S.BITS1.0   // 100-VEN-002 Enable
        [169].S.BITS1.1   // 100-VEN-002 Falla Resumen
        [169].S.BITS1.2   // 100-VEN-002 Conf. Marcha
        [169].S.BITS1.4   // 100-VEN-002 Cmd. Automatico
        [169].S.BITS1.26   // 100-VEN-002 FLL
        [169].S.BITS1.27   // 100-VEN-002 FV0
        [169].S.BITS1.28   // 100-VEN-002 FATO
        [169].S.BITS1.30   // 100-VEN-002 Falla Partida
        [169].S.BITS2.27   // 100-VEN-002 Cmd. Marcha
        [169].S.BITS2.20   // 100-VEN-002 Reset Falla
        [169].S.BITS2.23   // 100-VEN-002 Test
        [169].S.BITS2.30   // 100-VEN-002 OUT MARCHA
        [172].S.BITS1.27   // 100-TOR-001 FV0
        [171].S.BITS1.8   // 100-BIN-001 LL
        [171].S.BITS1.9   // 100-BIN-001 LM
        [171].S.BITS1.10   // 100-BIN-001 LH
        [172].S.BITS1.0   // 100-TOR-001 Enable
        [172].S.BITS1.1   // 100-TOR-001 Falla Resumen
        [172].S.BITS1.2   // 100-TOR-001 Conf. Marcha
        [172].S.BITS1.4   // 100-TOR-001 Cmd. Automatico
        [172].S.BITS1.26   // 100-TOR-001 FLL
        [172].S.BITS1.28   // 100-TOR-001 FATO
        [172].S.BITS1.30   // 100-TOR-001 Falla Partida
        [172].S.BITS2.27   // 100-TOR-001 Cmd. Marcha
        [172].S.BITS2.20   // 100-TOR-001 Reset Falla
        [172].S.BITS2.23   // 100-TOR-001 Test
        [172].S.BITS2.30   // 100-TOR-001 OUT MARCHA
        [178].S.BITS1.27   // 100-TOR-003 FV0
        [177].S.BITS1.8   // 100-BIN-003 LL
        [177].S.BITS1.9   // 100-BIN-003 LM
        [177].S.BITS1.10   // 100-BIN-003 LH
        [178].S.BITS1.0   // 100-TOR-003 Enable
        [178].S.BITS1.1   // 100-TOR-003 Falla Resumen
        [178].S.BITS1.2   // 100-TOR-003 Conf. Marcha
        [178].S.BITS1.4   // 100-TOR-003 Cmd. Automatico
        [178].S.BITS1.26   // 100-TOR-003 FLL
        [178].S.BITS1.28   // 100-TOR-003 FATO
        [178].S.BITS1.30   // 100-TOR-003 Falla Partida
        [178].S.BITS2.27   // 100-TOR-003 Cmd. Marcha
        [178].S.BITS2.20   // 100-TOR-003 Reset Falla
        [178].S.BITS2.23   // 100-TOR-003 Test
        [178].S.BITS2.30   // 100-TOR-003 OUT MARCHA
        [182].S.BITS1.0   // 100-TOR-037 Enable
        [182].S.BITS1.1   // 100-TOR-037 Falla Resumen
        [182].S.BITS1.2   // 100-TOR-037 Conf. Marcha
        [182].S.BITS1.4   // 100-TOR-037 Cmd. Automatico
        [182].S.BITS1.26   // 100-TOR-037 FLL
        [182].S.BITS1.27   // 100-TOR-037 FV0
        [182].S.BITS1.28   // 100-TOR-037 FATO
        [182].S.BITS1.30   // 100-TOR-037 Falla Partida
        [182].S.BITS2.27   // 100-TOR-037 Cmd. Marcha
        [182].S.BITS2.20   // 100-TOR-037 Reset Falla
        [182].S.BITS2.23   // 100-TOR-037 Test
        [182].S.BITS2.30   // 100-TOR-037 OUT MARCHA
        [184].S.BITS1.27   // 100-TOR-005 FV0
        [183].S.BITS1.8   // 100-BIN-005 LL
        [183].S.BITS1.9   // 100-BIN-005 LM
        [183].S.BITS1.10   // 100-BIN-005 LH
        [184].S.BITS1.0   // 100-TOR-005 Enable
        [184].S.BITS1.1   // 100-TOR-005 Falla Resumen
        [184].S.BITS1.2   // 100-TOR-005 Conf. Marcha
        [184].S.BITS1.4   // 100-TOR-005 Cmd. Automatico
        [184].S.BITS1.26   // 100-TOR-005 FLL
        [184].S.BITS1.28   // 100-TOR-005 FATO
        [184].S.BITS1.30   // 100-TOR-005 Falla Partida
        [184].S.BITS2.27   // 100-TOR-005 Cmd. Marcha
        [184].S.BITS2.20   // 100-TOR-005 Reset Falla
        [184].S.BITS2.23   // 100-TOR-005 Test
        [184].S.BITS2.30   // 100-TOR-005 OUT MARCHA
        [196].S.BITS1.27   // 100-TOR-008 FV0
        [195].S.BITS1.9   // 100-BIN-008 LM
        [196].S.BITS1.0   // 100-TOR-008 Enable
        [196].S.BITS1.1   // 100-TOR-008 Falla Resumen
        [196].S.BITS1.2   // 100-TOR-008 Conf. Marcha
        [196].S.BITS1.4   // 100-TOR-008 Cmd. Automatico
        [196].S.BITS1.26   // 100-TOR-008 FLL
        [196].S.BITS1.28   // 100-TOR-008 FATO
        [196].S.BITS1.30   // 100-TOR-008 Falla Partida
        [196].S.BITS2.27   // 100-TOR-008 Cmd. Marcha
        [196].S.BITS2.20   // 100-TOR-008 Reset Falla
        [196].S.BITS2.23   // 100-TOR-008 Test
        [196].S.BITS2.30   // 100-TOR-008 OUT MARCHA
        [199].S.BITS1.27   // 100-TOR-009 FV0
        [198].S.BITS1.8   // 100-BIN-009 LL
        [198].S.BITS1.9   // 100-BIN-009 LM
        [198].S.BITS1.10   // 100-BIN-009 LH
        [199].S.BITS1.0   // 100-TOR-009 Enable
        [199].S.BITS1.1   // 100-TOR-009 Falla Resumen
        [199].S.BITS1.2   // 100-TOR-009 Conf. Marcha
        [199].S.BITS1.4   // 100-TOR-009 Cmd. Automatico
        [199].S.BITS1.26   // 100-TOR-009 FLL
        [199].S.BITS1.28   // 100-TOR-009 FATO
        [199].S.BITS1.30   // 100-TOR-009 Falla Partida
        [199].S.BITS2.27   // 100-TOR-009 Cmd. Marcha
        [199].S.BITS2.20   // 100-TOR-009 Reset Falla
        [199].S.BITS2.23   // 100-TOR-009 Test
        [199].S.BITS2.30   // 100-TOR-009 OUT MARCHA
        [202].S.BITS1.27   // 7-RED-1171 FV0
        [201].S.BITS1.9   // 100-BIN-010 LM
        [202].S.BITS1.0   // 7-RED-1171 Enable
        [202].S.BITS1.1   // 7-RED-1171 Falla Resumen
        [202].S.BITS1.2   // 7-RED-1171 Conf. Marcha
        [202].S.BITS1.4   // 7-RED-1171 Cmd. Automatico
        [202].S.BITS1.26   // 7-RED-1171 FLL
        [202].S.BITS1.28   // 7-RED-1171 FATO
        [202].S.BITS1.30   // 7-RED-1171 Falla Partida
        [202].S.BITS2.27   // 7-RED-1171 Cmd. Marcha
        [202].S.BITS2.20   // 7-RED-1171 Reset Falla
        [202].S.BITS2.23   // 7-RED-1171 Test
        [202].S.BITS2.30   // 7-RED-1171 OUT MARCHA
        [205].S.BITS1.27   // 100-TOR-036 FV0
        [204].S.BITS1.8   // 100-BIN-011 LL
        [205].S.BITS1.0   // 100-TOR-036 Enable
        [205].S.BITS1.1   // 100-TOR-036 Falla Resumen
        [205].S.BITS1.2   // 100-TOR-036 Conf. Marcha
        [205].S.BITS1.4   // 100-TOR-036 Cmd. Automatico
        [205].S.BITS1.26   // 100-TOR-036 FLL
        [205].S.BITS1.28   // 100-TOR-036 FATO
        [205].S.BITS1.30   // 100-TOR-036 Falla Partida
        [205].S.BITS2.27   // 100-TOR-036 Cmd. Marcha
        [205].S.BITS2.20   // 100-TOR-036 Reset Falla
        [205].S.BITS2.23   // 100-TOR-036 Test
        [205].S.BITS2.30   // 100-TOR-036 OUT MARCHA
        [208].S.BITS1.27   // 7-VRT-1175 FV0
        [207].S.BITS1.8   // 100-BIN-012 LL
        [208].S.BITS1.0   // 7-VRT-1175 Enable
        [208].S.BITS1.1   // 7-VRT-1175 Falla Resumen
        [208].S.BITS1.2   // 7-VRT-1175 Conf. Marcha
        [208].S.BITS1.4   // 7-VRT-1175 Cmd. Automatico
        [208].S.BITS1.26   // 7-VRT-1175 FLL
        [208].S.BITS1.28   // 7-VRT-1175 FATO
        [208].S.BITS1.30   // 7-VRT-1175 Falla Partida
        [208].S.BITS2.27   // 7-VRT-1175 Cmd. Marcha
        [208].S.BITS2.20   // 7-VRT-1175 Reset Falla
        [208].S.BITS2.23   // 7-VRT-1175 Test
        [208].S.BITS2.30   // 7-VRT-1175 OUT MARCHA
        [211].S.BITS1.27   // 7-RED-1178 FV0
        [211].S.BITS1.0   // 7-RED-1178 Enable
        [211].S.BITS1.1   // 7-RED-1178 Falla Resumen
        [211].S.BITS1.2   // 7-RED-1178 Conf. Marcha
        [211].S.BITS1.4   // 7-RED-1178 Cmd. Automatico
        [211].S.BITS1.26   // 7-RED-1178 FLL
        [211].S.BITS1.28   // 7-RED-1178 FATO
        [211].S.BITS1.30   // 7-RED-1178 Falla Partida
        [211].S.BITS2.27   // 7-RED-1178 Cmd. Marcha
        [211].S.BITS2.20   // 7-RED-1178 Reset Falla
        [211].S.BITS2.23   // 7-RED-1178 Test
        [211].S.BITS2.30   // 7-RED-1178 OUT MARCHA
        [214].S.BITS1.27   // 100-TOR-014 FV0
        [213].S.BITS1.8   // 100-BIN-014 LL
        [214].S.BITS1.0   // 100-TOR-014 Enable
        [214].S.BITS1.1   // 100-TOR-014 Falla Resumen
        [214].S.BITS1.2   // 100-TOR-014 Conf. Marcha
        [214].S.BITS1.4   // 100-TOR-014 Cmd. Automatico
        [214].S.BITS1.26   // 100-TOR-014 FLL
        [214].S.BITS1.28   // 100-TOR-014 FATO
        [214].S.BITS1.30   // 100-TOR-014 Falla Partida
        [214].S.BITS2.27   // 100-TOR-014 Cmd. Marcha
        [214].S.BITS2.20   // 100-TOR-014 Reset Falla
        [214].S.BITS2.23   // 100-TOR-014 Test
        [214].S.BITS2.30   // 100-TOR-014 OUT MARCHA
        [217].S.BITS1.27   // 100-TOR-015 FV0
        [217].S.BITS1.0   // 100-TOR-015 Enable
        [217].S.BITS1.1   // 100-TOR-015 Falla Resumen
        [217].S.BITS1.2   // 100-TOR-015 Conf. Marcha
        [217].S.BITS1.4   // 100-TOR-015 Cmd. Automatico
        [217].S.BITS1.26   // 100-TOR-015 FLL
        [217].S.BITS1.28   // 100-TOR-015 FATO
        [217].S.BITS1.30   // 100-TOR-015 Falla Partida
        [217].S.BITS2.27   // 100-TOR-015 Cmd. Marcha
        [217].S.BITS2.20   // 100-TOR-015 Reset Falla
        [217].S.BITS2.23   // 100-TOR-015 Test
        [217].S.BITS2.30   // 100-TOR-015 OUT MARCHA
        [218].S.BITS1.0   // 7-BBA-1179b Enable
        [218].S.BITS1.1   // 7-BBA-1179b Falla Resumen
        [218].S.BITS1.2   // 7-BBA-1179b Conf. Marcha
        [218].S.BITS1.4   // 7-BBA-1179b Cmd. Automatico
        [218].S.BITS1.26   // 7-BBA-1179b FLL
        [218].S.BITS1.27   // 7-BBA-1179b FV0
        [218].S.BITS1.28   // 7-BBA-1179b FATO
        [218].S.BITS1.30   // 7-BBA-1179b Falla Partida
        [218].S.BITS2.27   // 7-BBA-1179b Cmd. Marcha
        [218].S.BITS2.20   // 7-BBA-1179b Reset Falla
        [218].S.BITS2.23   // 7-BBA-1179b Test
        [218].S.BITS2.30   // 7-BBA-1179b OUT MARCHA
        [220].S.BITS1.27   // 100-TOR-011 FV0
        [219].S.BITS1.9   // 100-BIN-016 LM
        [220].S.BITS1.0   // 100-TOR-011 Enable
        [220].S.BITS1.1   // 100-TOR-011 Falla Resumen
        [220].S.BITS1.2   // 100-TOR-011 Conf. Marcha
        [220].S.BITS1.4   // 100-TOR-011 Cmd. Automatico
        [220].S.BITS1.26   // 100-TOR-011 FLL
        [220].S.BITS1.28   // 100-TOR-011 FATO
        [220].S.BITS1.30   // 100-TOR-011 Falla Partida
        [220].S.BITS2.27   // 100-TOR-011 Cmd. Marcha
        [220].S.BITS2.20   // 100-TOR-011 Reset Falla
        [220].S.BITS2.23   // 100-TOR-011 Test
        [220].S.BITS2.30   // 100-TOR-011 OUT MARCHA
        [223].S.BITS1.27   // 100-TOR-035 FV0
        [223].S.BITS1.0   // 100-TOR-035 Enable
        [223].S.BITS1.1   // 100-TOR-035 Falla Resumen
        [223].S.BITS1.2   // 100-TOR-035 Conf. Marcha
        [223].S.BITS1.4   // 100-TOR-035 Cmd. Automatico
        [223].S.BITS1.26   // 100-TOR-035 FLL
        [223].S.BITS1.28   // 100-TOR-035 FATO
        [223].S.BITS1.30   // 100-TOR-035 Falla Partida
        [223].S.BITS2.27   // 100-TOR-035 Cmd. Marcha
        [223].S.BITS2.20   // 100-TOR-035 Reset Falla
        [223].S.BITS2.23   // 100-TOR-035 Test
        [223].S.BITS2.30   // 100-TOR-035 OUT MARCHA
        [239].S.BITS1.1   // 7-CON-1192 Falla Resumen
        [231].S.BITS1.8   // 7-TOL-1185 LL
        [231].S.BITS1.9   // 7-TOL-1185 LM
        [231].S.BITS1.10   // 7-TOL-1185 LH
        [239].S.BITS1.27   // 100-MMA-001 FV0
        [239].S.BITS1.0   // 7-CON-1192 Enable
        [239].S.BITS1.4   // 7-CON-1192 Conf Pos Cerrar
        [239].S.BITS1.26   // 100-MMA-001 FLL
        [239].S.BITS1.28   // 100-MMA-001 FATO
        [239].S.BITS1.30   // 7-CON-1192 Falla Cerrar
        [239].S.BITS2.27   // 7-CON-1192 Cmd. Open
        [239].S.BITS2.20   // 7-CON-1192 Reset Falla
        [239].S.BITS2.23   // 7-CON-1192 Test
        [239].S.BITS2.30   // 7-CON-1192 OUT CLOSE
        [242].S.BITS1.1   // 7-CON-1195 Falla Resumen
        [240].S.BITS1.8   // 100-MMA-001-B LL
        [240].S.BITS1.9   // 100-MMA-001-B LM
        [240].S.BITS1.10   // 100-MMA-001-B LH
        [242].S.BITS1.27   // 100-TOR-021 FV0
        [242].S.BITS1.0   // 7-CON-1195 Enable
        [242].S.BITS1.4   // 7-CON-1195 Conf Pos Cerrar
        [242].S.BITS1.26   // 100-TOR-021 FLL
        [242].S.BITS1.28   // 100-TOR-021 FATO
        [242].S.BITS1.30   // 7-CON-1195 Falla Cerrar
        [242].S.BITS2.27   // 7-CON-1195 Cmd. Open
        [242].S.BITS2.20   // 7-CON-1195 Reset Falla
        [242].S.BITS2.23   // 7-CON-1195 Test
        [242].S.BITS2.30   // 7-CON-1195 OUT CLOSE
        [244].S.BITS1.27   // 7-ROS-1201 FV0
        [243].S.BITS1.9   // 100-TOL-007 LM
        [244].S.BITS1.0   // 7-ROS-1201 Enable
        [244].S.BITS1.1   // 7-ROS-1201 Falla Resumen
        [244].S.BITS1.2   // 7-ROS-1201 Conf. Marcha
        [244].S.BITS1.4   // 7-ROS-1201 Cmd. Automatico
        [244].S.BITS1.26   // 7-ROS-1201 FLL
        [244].S.BITS1.28   // 7-ROS-1201 FATO
        [244].S.BITS1.30   // 7-ROS-1201 Falla Partida
        [244].S.BITS2.27   // 7-ROS-1201 Cmd. Marcha
        [244].S.BITS2.20   // 7-ROS-1201 Reset Falla
        [244].S.BITS2.23   // 7-ROS-1201 Test
        [244].S.BITS2.30   // 7-ROS-1201 OUT MARCHA
        [246].S.BITS1.27   // 7-ROS-1203 FV0
        [245].S.BITS1.9   // 100-TOL-008 LM
        [246].S.BITS1.0   // 7-ROS-1203 Enable
        [246].S.BITS1.1   // 7-ROS-1203 Falla Resumen
        [246].S.BITS1.2   // 7-ROS-1203 Conf. Marcha
        [246].S.BITS1.4   // 7-ROS-1203 Cmd. Automatico
        [246].S.BITS1.26   // 7-ROS-1203 FLL
        [246].S.BITS1.28   // 7-ROS-1203 FATO
        [246].S.BITS1.30   // 7-ROS-1203 Falla Partida
        [246].S.BITS2.27   // 7-ROS-1203 Cmd. Marcha
        [246].S.BITS2.20   // 7-ROS-1203 Reset Falla
        [246].S.BITS2.23   // 7-ROS-1203 Test
        [246].S.BITS2.30   // 7-ROS-1203 OUT MARCHA
        [248].S.BITS1.27   // 7-MOL-1205 FV0
        [247].S.BITS1.9   // 7-TOL-1204 LM
        [248].S.BITS1.0   // 7-MOL-1205 Enable
        [248].S.BITS1.1   // 7-MOL-1205 Falla Resumen
        [248].S.BITS1.2   // 7-MOL-1205 Conf. Marcha
        [248].S.BITS1.4   // 7-MOL-1205 Cmd. Automatico
        [248].S.BITS1.26   // 7-MOL-1205 FLL
        [248].S.BITS1.28   // 7-MOL-1205 FATO
        [248].S.BITS1.30   // 7-MOL-1205 Falla Partida
        [248].S.BITS2.27   // 7-MOL-1205 Cmd. Marcha
        [248].S.BITS2.20   // 7-MOL-1205 Reset Falla
        [248].S.BITS2.23   // 7-MOL-1205 Test
        [248].S.BITS2.30   // 7-MOL-1205 OUT MARCHA
        [250].S.BITS1.27   // 100-TOR-017 FV0
        [250].S.BITS1.0   // 100-TOR-017 Enable
        [250].S.BITS1.1   // 100-TOR-017 Falla Resumen
        [250].S.BITS1.2   // 100-TOR-017 Conf. Marcha
        [250].S.BITS1.4   // 100-TOR-017 Cmd. Automatico
        [250].S.BITS1.26   // 100-TOR-017 FLL
        [250].S.BITS1.28   // 100-TOR-017 FATO
        [250].S.BITS1.30   // 100-TOR-017 Falla Partida
        [250].S.BITS2.27   // 100-TOR-017 Cmd. Marcha
        [250].S.BITS2.20   // 100-TOR-017 Reset Falla
        [250].S.BITS2.23   // 100-TOR-017 Test
        [250].S.BITS2.30   // 100-TOR-017 OUT MARCHA
        [252].S.BITS1.27   // 7-RED-004C FV0
        [252].S.BITS1.0   // 7-RED-004C Enable
        [252].S.BITS1.1   // 7-RED-004C Falla Resumen
        [252].S.BITS1.4   // 7-RED-004C Cmd. Automatico
        [252].S.BITS1.26   // 7-RED-004C FLL
        [252].S.BITS1.28   // 7-RED-004C FATO
        [252].S.BITS1.30   // 7-RED-004C Falla Partida
        [252].S.BITS2.27   // 7-RED-004C Cmd. Marcha
        [252].S.BITS2.20   // 7-RED-004C Reset Falla
        [252].S.BITS2.23   // 7-RED-004C Test
        [252].S.BITS2.30   // 7-RED-004C OUT MARCHA
        [255].S.BITS1.30   // 100-TOL-004-1 Falla Cerrar
        [254].S.BITS1.8   // 100-TOL-004 LL
        [254].S.BITS1.9   // 100-TOL-004 LM
        [254].S.BITS1.10   // 100-TOL-004 LH
        [255].S.BITS1.0   // 100-TOL-004-1 Enable
        [255].S.BITS1.1   // 100-TOL-004-1 Falla Resumen
        [255].S.BITS1.2   // 100-TOL-004-1 Conf Pos Abrir
        [255].S.BITS1.4   // 100-TOL-004-1 Conf Pos Cerrar
        [255].S.BITS1.29   // 100-TOL-004-1 Falla Abrir
        [255].S.BITS2.20   // 100-TOL-004-1 Reset Falla
        [255].S.BITS2.23   // 100-TOL-004-1 Test
        [255].S.BITS2.27   // 100-TOL-004-1 Cmd. Open
        [255].S.BITS2.30   // 100-TOL-004-1 OUT CLOSE
        [255].S.BITS2.31   // 100-TOL-004-1 OUT OPEN
        [262].S.BITS1.27   // 100-DOS-001-M01 FV0
        [261].S.BITS1.8   // 100-DOS-001-T01 LL
        [261].S.BITS1.9   // 100-DOS-001-T01 LM
        [261].S.BITS1.10   // 100-DOS-001-T01 LH
        [262].S.BITS1.0   // 100-DOS-001-M01 Enable
        [262].S.BITS1.1   // 100-DOS-001-M01 Falla Resumen
        [262].S.BITS1.2   // 100-DOS-001-M01 Conf. Marcha
        [262].S.BITS1.4   // 100-DOS-001-M01 Cmd. Automatico
        [262].S.BITS1.26   // 100-DOS-001-M01 FLL
        [262].S.BITS1.28   // 100-DOS-001-M01 FATO
        [262].S.BITS1.30   // 100-DOS-001-M01 Falla Partida
        [262].S.BITS2.27   // 100-DOS-001-M01 Cmd. Marcha
        [262].S.BITS2.20   // 100-DOS-001-M01 Reset Falla
        [262].S.BITS2.23   // 100-DOS-001-M01 Test
        [262].S.BITS2.30   // 100-DOS-001-M01 OUT MARCHA
        [264].S.BITS1.27   // 100-DOS-001-MO2 FV0
        [263].S.BITS1.8   // 100-DOS-001-TO2 LL
        [263].S.BITS1.9   // 100-DOS-001-TO2 LM
        [263].S.BITS1.10   // 100-DOS-001-TO2 LH
        [264].S.BITS1.0   // 100-DOS-001-MO2 Enable
        [264].S.BITS1.1   // 100-DOS-001-MO2 Falla Resumen
        [264].S.BITS1.2   // 100-DOS-001-MO2 Conf. Marcha
        [264].S.BITS1.4   // 100-DOS-001-MO2 Cmd. Automatico
        [264].S.BITS1.26   // 100-DOS-001-MO2 FLL
        [264].S.BITS1.28   // 100-DOS-001-MO2 FATO
        [264].S.BITS1.30   // 100-DOS-001-MO2 Falla Partida
        [264].S.BITS2.27   // 100-DOS-001-MO2 Cmd. Marcha
        [264].S.BITS2.20   // 100-DOS-001-MO2 Reset Falla
        [264].S.BITS2.23   // 100-DOS-001-MO2 Test
        [264].S.BITS2.30   // 100-DOS-001-MO2 OUT MARCHA
        [266].S.BITS1.27   // 100-DOS-001-M03 FV0
        [265].S.BITS1.8   // 100-DOS-001-T03 LL
        [265].S.BITS1.9   // 100-DOS-001-T03 LM
        [265].S.BITS1.10   // 100-DOS-001-T03 LH
        [266].S.BITS1.0   // 100-DOS-001-M03 Enable
        [266].S.BITS1.1   // 100-DOS-001-M03 Falla Resumen
        [266].S.BITS1.2   // 100-DOS-001-M03 Conf. Marcha
        [266].S.BITS1.4   // 100-DOS-001-M03 Cmd. Automatico
        [266].S.BITS1.26   // 100-DOS-001-M03 FLL
        [266].S.BITS1.28   // 100-DOS-001-M03 FATO
        [266].S.BITS1.30   // 100-DOS-001-M03 Falla Partida
        [266].S.BITS2.27   // 100-DOS-001-M03 Cmd. Marcha
        [266].S.BITS2.20   // 100-DOS-001-M03 Reset Falla
        [266].S.BITS2.23   // 100-DOS-001-M03 Test
        [266].S.BITS2.30   // 100-DOS-001-M03 OUT MARCHA
        [268].S.BITS1.27   // 100-DOS-001-M04 FV0
        [267].S.BITS1.8   // 100-DOS-001-T04 LL
        [267].S.BITS1.9   // 100-DOS-001-T04 LM
        [267].S.BITS1.10   // 100-DOS-001-T04 LH
        [268].S.BITS1.0   // 100-DOS-001-M04 Enable
        [268].S.BITS1.1   // 100-DOS-001-M04 Falla Resumen
        [268].S.BITS1.2   // 100-DOS-001-M04 Conf. Marcha
        [268].S.BITS1.4   // 100-DOS-001-M04 Cmd. Automatico
        [268].S.BITS1.26   // 100-DOS-001-M04 FLL
        [268].S.BITS1.28   // 100-DOS-001-M04 FATO
        [268].S.BITS1.30   // 100-DOS-001-M04 Falla Partida
        [268].S.BITS2.27   // 100-DOS-001-M04 Cmd. Marcha
        [268].S.BITS2.20   // 100-DOS-001-M04 Reset Falla
        [268].S.BITS2.23   // 100-DOS-001-M04 Test
        [268].S.BITS2.30   // 100-DOS-001-M04 OUT MARCHA
        [270].S.BITS1.27   // 100-DOS-001-M05 FV0
        [269].S.BITS1.8   // 100-DOS-001-T05 LL
        [269].S.BITS1.9   // 100-DOS-001-T05 LM
        [269].S.BITS1.10   // 100-DOS-001-T05 LH
        [270].S.BITS1.0   // 100-DOS-001-M05 Enable
        [270].S.BITS1.1   // 100-DOS-001-M05 Falla Resumen
        [270].S.BITS1.2   // 100-DOS-001-M05 Conf. Marcha
        [270].S.BITS1.4   // 100-DOS-001-M05 Cmd. Automatico
        [270].S.BITS1.26   // 100-DOS-001-M05 FLL
        [270].S.BITS1.28   // 100-DOS-001-M05 FATO
        [270].S.BITS1.30   // 100-DOS-001-M05 Falla Partida
        [270].S.BITS2.27   // 100-DOS-001-M05 Cmd. Marcha
        [270].S.BITS2.20   // 100-DOS-001-M05 Reset Falla
        [270].S.BITS2.23   // 100-DOS-001-M05 Test
        [270].S.BITS2.30   // 100-DOS-001-M05 OUT MARCHA
        [272].S.BITS1.27   // 100-DOS-001-M06 FV0
        [271].S.BITS1.8   // 100-DOS-001-T06 LL
        [271].S.BITS1.9   // 100-DOS-001-T06 LM
        [271].S.BITS1.10   // 100-DOS-001-T06 LH
        [272].S.BITS1.0   // 100-DOS-001-M06 Enable
        [272].S.BITS1.1   // 100-DOS-001-M06 Falla Resumen
        [272].S.BITS1.2   // 100-DOS-001-M06 Conf. Marcha
        [272].S.BITS1.4   // 100-DOS-001-M06 Cmd. Automatico
        [272].S.BITS1.26   // 100-DOS-001-M06 FLL
        [272].S.BITS1.28   // 100-DOS-001-M06 FATO
        [272].S.BITS1.30   // 100-DOS-001-M06 Falla Partida
        [272].S.BITS2.27   // 100-DOS-001-M06 Cmd. Marcha
        [272].S.BITS2.20   // 100-DOS-001-M06 Reset Falla
        [272].S.BITS2.23   // 100-DOS-001-M06 Test
        [272].S.BITS2.30   // 100-DOS-001-M06 OUT MARCHA
        [274].S.BITS1.27   // 100-DOS-001-M07 FV0
        [273].S.BITS1.8   // 100-D0S-001-T07 LL
        [273].S.BITS1.9   // 100-D0S-001-T07 LM
        [273].S.BITS1.10   // 100-D0S-001-T07 LH
        [274].S.BITS1.0   // 100-DOS-001-M07 Enable
        [274].S.BITS1.1   // 100-DOS-001-M07 Falla Resumen
        [274].S.BITS1.2   // 100-DOS-001-M07 Conf. Marcha
        [274].S.BITS1.4   // 100-DOS-001-M07 Cmd. Automatico
        [274].S.BITS1.26   // 100-DOS-001-M07 FLL
        [274].S.BITS1.28   // 100-DOS-001-M07 FATO
        [274].S.BITS1.30   // 100-DOS-001-M07 Falla Partida
        [274].S.BITS2.27   // 100-DOS-001-M07 Cmd. Marcha
        [274].S.BITS2.20   // 100-DOS-001-M07 Reset Falla
        [274].S.BITS2.23   // 100-DOS-001-M07 Test
        [274].S.BITS2.30   // 100-DOS-001-M07 OUT MARCHA
        [276].S.BITS1.27   // 100-DOS-001-M08 FV0
        [275].S.BITS1.8   // 100-DOS-001-T08 LL
        [275].S.BITS1.9   // 100-DOS-001-T08 LM
        [275].S.BITS1.10   // 100-DOS-001-T08 LH
        [276].S.BITS1.0   // 100-DOS-001-M08 Enable
        [276].S.BITS1.1   // 100-DOS-001-M08 Falla Resumen
        [276].S.BITS1.2   // 100-DOS-001-M08 Conf. Marcha
        [276].S.BITS1.4   // 100-DOS-001-M08 Cmd. Automatico
        [276].S.BITS1.26   // 100-DOS-001-M08 FLL
        [276].S.BITS1.28   // 100-DOS-001-M08 FATO
        [276].S.BITS1.30   // 100-DOS-001-M08 Falla Partida
        [276].S.BITS2.27   // 100-DOS-001-M08 Cmd. Marcha
        [276].S.BITS2.20   // 100-DOS-001-M08 Reset Falla
        [276].S.BITS2.23   // 100-DOS-001-M08 Test
        [276].S.BITS2.30   // 100-DOS-001-M08 OUT MARCHA
        [278].S.BITS1.27   // 100-DOS-001-M09 FV0
        [277].S.BITS1.8   // 100-DOS-001-T09 LL
        [277].S.BITS1.9   // 100-DOS-001-T09 LM
        [277].S.BITS1.10   // 100-DOS-001-T09 LH
        [278].S.BITS1.0   // 100-DOS-001-M09 Enable
        [278].S.BITS1.1   // 100-DOS-001-M09 Falla Resumen
        [278].S.BITS1.2   // 100-DOS-001-M09 Conf. Marcha
        [278].S.BITS1.4   // 100-DOS-001-M09 Cmd. Automatico
        [278].S.BITS1.26   // 100-DOS-001-M09 FLL
        [278].S.BITS1.28   // 100-DOS-001-M09 FATO
        [278].S.BITS1.30   // 100-DOS-001-M09 Falla Partida
        [278].S.BITS2.27   // 100-DOS-001-M09 Cmd. Marcha
        [278].S.BITS2.20   // 100-DOS-001-M09 Reset Falla
        [278].S.BITS2.23   // 100-DOS-001-M09 Test
        [278].S.BITS2.30   // 100-DOS-001-M09 OUT MARCHA
        [280].S.BITS1.27   // 100-DOS-100-M10 FV0
        [279].S.BITS1.8   // 100-DOS-100-T10 LL
        [279].S.BITS1.9   // 100-DOS-100-T10 LM
        [279].S.BITS1.10   // 100-DOS-100-T10 LH
        [280].S.BITS1.0   // 100-DOS-100-M10 Enable
        [280].S.BITS1.1   // 100-DOS-100-M10 Falla Resumen
        [280].S.BITS1.2   // 100-DOS-100-M10 Conf. Marcha
        [280].S.BITS1.4   // 100-DOS-100-M10 Cmd. Automatico
        [280].S.BITS1.26   // 100-DOS-100-M10 FLL
        [280].S.BITS1.28   // 100-DOS-100-M10 FATO
        [280].S.BITS1.30   // 100-DOS-100-M10 Falla Partida
        [280].S.BITS2.27   // 100-DOS-100-M10 Cmd. Marcha
        [280].S.BITS2.20   // 100-DOS-100-M10 Reset Falla
        [280].S.BITS2.23   // 100-DOS-100-M10 Test
        [280].S.BITS2.30   // 100-DOS-100-M10 OUT MARCHA
        [282].S.BITS1.27   // 100-DOS-100-M11 FV0
        [281].S.BITS1.8   // 100-DOS-100-T11 LL
        [281].S.BITS1.9   // 100-DOS-100-T11 LM
        [281].S.BITS1.10   // 100-DOS-100-T11 LH
        [282].S.BITS1.0   // 100-DOS-100-M11 Enable
        [282].S.BITS1.1   // 100-DOS-100-M11 Falla Resumen
        [282].S.BITS1.2   // 100-DOS-100-M11 Conf. Marcha
        [282].S.BITS1.4   // 100-DOS-100-M11 Cmd. Automatico
        [282].S.BITS1.26   // 100-DOS-100-M11 FLL
        [282].S.BITS1.28   // 100-DOS-100-M11 FATO
        [282].S.BITS1.30   // 100-DOS-100-M11 Falla Partida
        [282].S.BITS2.27   // 100-DOS-100-M11 Cmd. Marcha
        [282].S.BITS2.20   // 100-DOS-100-M11 Reset Falla
        [282].S.BITS2.23   // 100-DOS-100-M11 Test
        [282].S.BITS2.30   // 100-DOS-100-M11 OUT MARCHA
        [284].S.BITS1.27   // 100-DOS-100-M12 FV0
        [283].S.BITS1.8   // 100-DOS-100-T12 LL
        [283].S.BITS1.9   // 100-DOS-100-T12 LM
        [283].S.BITS1.10   // 100-DOS-100-T12 LH
        [284].S.BITS1.0   // 100-DOS-100-M12 Enable
        [284].S.BITS1.1   // 100-DOS-100-M12 Falla Resumen
        [284].S.BITS1.2   // 100-DOS-100-M12 Conf. Marcha
        [284].S.BITS1.4   // 100-DOS-100-M12 Cmd. Automatico
        [284].S.BITS1.26   // 100-DOS-100-M12 FLL
        [284].S.BITS1.28   // 100-DOS-100-M12 FATO
        [284].S.BITS1.30   // 100-DOS-100-M12 Falla Partida
        [284].S.BITS2.27   // 100-DOS-100-M12 Cmd. Marcha
        [284].S.BITS2.20   // 100-DOS-100-M12 Reset Falla
        [284].S.BITS2.23   // 100-DOS-100-M12 Test
        [284].S.BITS2.30   // 100-DOS-100-M12 OUT MARCHA
        [289].S.BITS1.27   // 100-TDP-003 FV0
        [287].S.BITS1.8   // 100-DOS-001-T LL
        [287].S.BITS1.9   // 100-DOS-001-T LM
        [287].S.BITS1.10   // 100-DOS-001-T LH
        [289].S.BITS1.0   // 100-TDP-003 Enable
        [289].S.BITS1.1   // 100-TDP-003 Falla Resumen
        [289].S.BITS1.4   // 100-TDP-003 Cmd. Automatico
        [289].S.BITS1.26   // 100-TDP-003 FLL
        [289].S.BITS1.28   // 100-TDP-003 FATO
        [289].S.BITS1.30   // 100-TDP-003 Falla Partida
        [289].S.BITS2.27   // 100-TDP-003 Cmd. Marcha
        [289].S.BITS2.20   // 100-TDP-003 Reset Falla
        [289].S.BITS2.23   // 100-TDP-003 Test
        [289].S.BITS2.30   // 100-TDP-003 OUT MARCHA
        [292].S.BITS1.26   // 100-TDP-004 FLL
        [292].S.BITS1.27   // 100-TDP-004 FV0
        [292].S.BITS1.28   // 100-TDP-004 FATO
        [293].S.BITS1.2   // 100-ELV-002 Conf. Marcha
        [293].S.BITS1.26   // 100-ELV-002 FLL
        [293].S.BITS1.27   // 100-ELV-002 FV0
        [293].S.BITS1.28   // 100-ELV-002 FATO
        [293].S.BITS2.27   // 100-ELV-002 Cmd. Marcha
        [294].S.BITS1.0   // 100-TDP-005 Enable
        [294].S.BITS1.1   // 100-TDP-005 Falla Resumen
        [294].S.BITS1.26   // 100-TDP-005 FLL
        [294].S.BITS1.27   // 100-TDP-005 FV0
        [294].S.BITS1.28   // 100-TDP-005 FATO
        [294].S.BITS2.20   // 100-TDP-005 Reset Falla
        [294].S.BITS2.23   // 100-TDP-005 Test
        [299].S.BITS1.27   // 100-TDP-006 FV0
        [296].S.BITS1.8   // 100-TOL-003 LL
        [296].S.BITS1.9   // 100-TOL-003 LM
        [296].S.BITS1.10   // 100-TOL-003 LH
        [299].S.BITS1.0   // 100-TDP-006 Enable
        [299].S.BITS1.1   // 100-TDP-006 Falla Resumen
        [299].S.BITS1.2   // 100-TDP-006 Conf. Marcha
        [299].S.BITS1.4   // 100-TDP-006 Cmd. Automatico
        [299].S.BITS1.26   // 100-TDP-006 FLL
        [299].S.BITS1.28   // 100-TDP-006 FATO
        [299].S.BITS1.30   // 100-TDP-006 Falla Partida
        [299].S.BITS2.27   // 100-TDP-006 Cmd. Marcha
        [299].S.BITS2.20   // 100-TDP-006 Reset Falla
        [299].S.BITS2.23   // 100-TDP-006 Test
        [299].S.BITS2.30   // 100-TDP-006 OUT MARCHA
        [302].S.BITS1.27   // 100-BCE-003 FV0
        [301].S.BITS1.8   // 8-TOL-600 LL
        [301].S.BITS1.9   // 8-TOL-600 LM
        [301].S.BITS1.10   // 8-TOL-600 LH
        [302].S.BITS1.0   // 100-BCE-003 Enable
        [302].S.BITS1.1   // 100-BCE-003 Falla Resumen
        [302].S.BITS1.2   // 100-BCE-003 Conf. Marcha
        [302].S.BITS1.4   // 100-BCE-003 Cmd. Automatico
        [302].S.BITS1.26   // 100-BCE-003 FLL
        [302].S.BITS1.28   // 100-BCE-003 FATO
        [302].S.BITS1.30   // 100-BCE-003 Falla Partida
        [302].S.BITS2.27   // 100-BCE-003 Cmd. Marcha
        [302].S.BITS2.20   // 100-BCE-003 Reset Falla
        [302].S.BITS2.23   // 100-BCE-003 Test
        [302].S.BITS2.30   // 100-BCE-003 OUT MARCHA
        [303].S.BITS1.26   // XY-6170 FLL
        [303].S.BITS1.27   // XY-6170 FV0
        [303].S.BITS1.28   // XY-6170 FATO
        [304].S.BITS1.0   // 100-BCE-005 Enable
        [304].S.BITS1.1   // 100-BCE-005 Falla Resumen
        [304].S.BITS1.4   // 100-BCE-005 Cmd. Automatico
        [304].S.BITS1.26   // 100-BCE-005 FLL
        [304].S.BITS1.27   // 100-BCE-005 FV0
        [304].S.BITS1.28   // 100-BCE-005 FATO
        [304].S.BITS1.30   // 100-BCE-005 Falla Partida
        [304].S.BITS2.27   // 100-BCE-005 Cmd. Marcha
        [304].S.BITS2.20   // 100-BCE-005 Reset Falla
        [304].S.BITS2.23   // 100-BCE-005 Test
        [304].S.BITS2.30   // 100-BCE-005 OUT MARCHA
        [308].S.BITS1.27   // 8-ROS-614 FV0
        [307].S.BITS1.8   // 8-TOL-612 LL
        [307].S.BITS1.9   // 8-TOL-612 LM
        [307].S.BITS1.10   // 8-TOL-612 LH
        [308].S.BITS1.0   // 8-ROS-614 Enable
        [308].S.BITS1.1   // 8-ROS-614 Falla Resumen
        [308].S.BITS1.2   // 8-ROS-614 Conf. Marcha
        [308].S.BITS1.4   // 8-ROS-614 Cmd. Automatico
        [308].S.BITS1.26   // 8-ROS-614 FLL
        [308].S.BITS1.28   // 8-ROS-614 FATO
        [308].S.BITS1.30   // 8-ROS-614 Falla Partida
        [308].S.BITS2.27   // 8-ROS-614 Cmd. Marcha
        [308].S.BITS2.20   // 8-ROS-614 Reset Falla
        [308].S.BITS2.23   // 8-ROS-614 Test
        [308].S.BITS2.30   // 8-ROS-614 OUT MARCHA
        [311].S.BITS1.8   // 100-UDO-003 LL
        [311].S.BITS1.9   // 100-UDO-003 LM
        [311].S.BITS1.10   // 100-UDO-003 LH
        [313].S.BITS1.26   // XY-6102 FLL
        [313].S.BITS1.27   // XY-6102 FV0
        [313].S.BITS1.28   // XY-6102 FATO
        [314].S.BITS1.0   // 8-VRT-629 Enable
        [314].S.BITS1.1   // 8-VRT-629 Falla Resumen
        [314].S.BITS1.2   // 8-VRT-629 Conf. Marcha
        [314].S.BITS1.4   // 8-VRT-629 Cmd. Automatico
        [314].S.BITS1.26   // 8-VRT-629 FLL
        [314].S.BITS1.27   // 8-VRT-629 FV0
        [314].S.BITS1.28   // 8-VRT-629 FATO
        [314].S.BITS1.30   // 8-VRT-629 Falla Partida
        [314].S.BITS2.27   // 8-VRT-629 Cmd. Marcha
        [314].S.BITS2.20   // 8-VRT-629 Reset Falla
        [314].S.BITS2.23   // 8-VRT-629 Test
        [314].S.BITS2.30   // 8-VRT-629 OUT MARCHA
        [315].S.BITS1.0   // 8-ENF-630-1 Enable
        [315].S.BITS1.1   // 8-ENF-630-1 Falla Resumen
        [315].S.BITS1.2   // 8-ENF-630-1 Conf. Marcha
        [315].S.BITS1.4   // 8-ENF-630-1 Cmd. Automatico
        [315].S.BITS1.26   // 8-ENF-630-1 FLL
        [315].S.BITS1.27   // 8-ENF-630-1 FV0
        [315].S.BITS1.28   // 8-ENF-630-1 FATO
        [315].S.BITS1.30   // 8-ENF-630-1 Falla Partida
        [315].S.BITS2.27   // 8-ENF-630-1 Cmd. Marcha
        [315].S.BITS2.20   // 8-ENF-630-1 Reset Falla
        [315].S.BITS2.23   // 8-ENF-630-1 Test
        [315].S.BITS2.30   // 8-ENF-630-1 OUT MARCHA
        [316].S.BITS1.0   // 100-VEN-LICINA-1 Enable
        [316].S.BITS1.1   // 100-VEN-LICINA-1 Falla Resumen
        [316].S.BITS1.2   // 100-VEN-LICINA-1 Conf. Marcha
        [316].S.BITS1.4   // 100-VEN-LICINA-1 Cmd. Automatico
        [316].S.BITS1.26   // 100-VEN-LICINA-1 FLL
        [316].S.BITS1.27   // 100-VEN-LICINA-1 FV0
        [316].S.BITS1.28   // 100-VEN-LICINA-1 FATO
        [316].S.BITS1.30   // 100-VEN-LICINA-1 Falla Partida
        [316].S.BITS2.27   // 100-VEN-LICINA-1 Cmd. Marcha
        [316].S.BITS2.20   // 100-VEN-LICINA-1 Reset Falla
        [316].S.BITS2.23   // 100-VEN-LICINA-1 Test
        [316].S.BITS2.30   // 100-VEN-LICINA-1 OUT MARCHA
        [317].S.BITS1.0   // 8-ENF-630-2 Enable
        [317].S.BITS1.1   // 8-ENF-630-2 Falla Resumen
        [317].S.BITS1.2   // 8-ENF-630-2 Conf. Marcha
        [317].S.BITS1.4   // 8-ENF-630-2 Cmd. Automatico
        [317].S.BITS1.26   // 8-ENF-630-2 FLL
        [317].S.BITS1.27   // 8-ENF-630-2 FV0
        [317].S.BITS1.28   // 8-ENF-630-2 FATO
        [317].S.BITS1.30   // 8-ENF-630-2 Falla Partida
        [317].S.BITS2.27   // 8-ENF-630-2 Cmd. Marcha
        [317].S.BITS2.20   // 8-ENF-630-2 Reset Falla
        [317].S.BITS2.23   // 8-ENF-630-2 Test
        [317].S.BITS2.30   // 8-ENF-630-2 OUT MARCHA
        [322].S.BITS1.27   // 8-VEN-637 FV0
        [321].S.BITS1.8   // 100-MIX-001-T LL
        [321].S.BITS1.9   // 100-MIX-001-T LM
        [321].S.BITS1.10   // 100-MIX-001-T LH
        [322].S.BITS1.0   // 8-VEN-637 Enable
        [322].S.BITS1.1   // 8-VEN-637 Falla Resumen
        [322].S.BITS1.2   // 8-VEN-637 Conf. Marcha
        [322].S.BITS1.4   // 8-VEN-637 Cmd. Automatico
        [322].S.BITS1.26   // 8-VEN-637 FLL
        [322].S.BITS1.28   // 8-VEN-637 FATO
        [322].S.BITS1.30   // 8-VEN-637 Falla Partida
        [322].S.BITS2.27   // 8-VEN-637 Cmd. Marcha
        [322].S.BITS2.20   // 8-VEN-637 Reset Falla
        [322].S.BITS2.23   // 8-VEN-637 Test
        [322].S.BITS2.30   // 8-VEN-637 OUT MARCHA
        [324].S.BITS1.2   // 8-VRT-639 Conf. Marcha
        [324].S.BITS1.29   // XY-6103 Falla Abrir
        [324].S.BITS2.31   // XY-6103 OUT OPEN
        [334].S.BITS1.0   // 8-ROS-652 Enable
        [334].S.BITS1.1   // 8-ROS-652 Falla Resumen
        [334].S.BITS1.2   // 8-ROS-652 Conf. Marcha
        [334].S.BITS1.4   // 8-ROS-652 Cmd. Automatico
        [334].S.BITS1.26   // 8-ROS-652 FLL
        [334].S.BITS1.27   // 8-ROS-652 FV0
        [334].S.BITS1.28   // 8-ROS-652 FATO
        [334].S.BITS1.30   // 8-ROS-652 Falla Partida
        [334].S.BITS2.27   // 8-ROS-652 Cmd. Marcha
        [334].S.BITS2.20   // 8-ROS-652 Reset Falla
        [334].S.BITS2.23   // 8-ROS-652 Test
        [334].S.BITS2.30   // 8-ROS-652 OUT MARCHA
        [337].S.BITS1.0   // 8-RED-658 Enable
        [337].S.BITS1.1   // 8-RED-658 Falla Resumen
        [337].S.BITS1.2   // 8-RED-658 Conf. Marcha
        [337].S.BITS1.4   // 8-RED-658 Cmd. Automatico
        [337].S.BITS1.26   // 8-RED-658 FLL
        [337].S.BITS1.27   // 8-RED-658 FV0
        [337].S.BITS1.28   // 8-RED-658 FATO
        [337].S.BITS1.30   // 8-RED-658 Falla Partida
        [337].S.BITS2.27   // 8-RED-658 Cmd. Marcha
        [337].S.BITS2.20   // 8-RED-658 Reset Falla
        [337].S.BITS2.23   // 8-RED-658 Test
        [337].S.BITS2.30   // 8-RED-658 OUT MARCHA
        [344].S.BITS1.30   // 110-LMG-001-01 Falla Cerrar
        [343].S.BITS1.8   // 8-TOL-700 LL
        [343].S.BITS1.9   // 8-TOL-700 LM
        [343].S.BITS1.10   // 8-TOL-700 LH
        [344].S.BITS1.0   // 110-LMG-001-01 Enable
        [344].S.BITS1.1   // 110-LMG-001-01 Falla Resumen
        [344].S.BITS1.2   // 110-LMG-001-01 Conf Pos Abrir
        [344].S.BITS1.4   // 110-LMG-001-01 Conf Pos Cerrar
        [344].S.BITS1.29   // 110-LMG-001-01 Falla Abrir
        [344].S.BITS2.20   // 110-LMG-001-01 Reset Falla
        [344].S.BITS2.23   // 110-LMG-001-01 Test
        [344].S.BITS2.30   // 110-LMG-001-01 OUT CLOSE
        [344].S.BITS2.31   // 110-LMG-001-01 OUT OPEN
        [346].S.BITS1.2   // 110-LMG-002 Conf. Pos. Izquierda
        [346].S.BITS1.4   // 110-LMG-002 Conf. Pos. Derecha
        [346].S.BITS1.29   // 110-LMG-002 Falla Pos. Izquierda
        [346].S.BITS1.30   // 110-LMG-002 Falla Pos. Derecha
        [346].S.BITS2.26   // 110-LMG-002 Cmd. Pos . Izquierda
        [346].S.BITS2.27   // 110-LMG-002 Cmd. Pos. Derecha
        [346].S.BITS2.30   // 110-LMG-002 Out Izquierda
        [346].S.BITS2.31   // 110-LMG-002 Out Derecha
        [347].S.BITS1.8   // 8-TOL-708 LL
        [347].S.BITS1.9   // 8-TOL-708 LM
        [347].S.BITS1.10   // 8-TOL-708 LH
        [349].S.BITS1.27   // 110-LRT-001 FV0
        [349].S.BITS1.26   // 110-LRT-001 FLL
        [349].S.BITS1.28   // 110-LRT-001 FATO
        [351].S.BITS1.27   // 8-ACO-716 FV0
        [351].S.BITS1.26   // 8-ACO-716 FLL
        [351].S.BITS1.28   // 8-ACO-716 FATO
        [352].S.BITS1.0   // 8-FPR-718 Enable
        [352].S.BITS1.1   // 8-FPR-718 Falla Resumen
        [352].S.BITS1.2   // 8-FPR-718 Conf. Marcha
        [352].S.BITS1.4   // 8-FPR-718 Cmd. Automatico
        [352].S.BITS1.26   // 8-FPR-718 FLL
        [352].S.BITS1.27   // 8-FPR-718 FV0
        [352].S.BITS1.28   // 8-FPR-718 FATO
        [352].S.BITS1.30   // 8-FPR-718 Falla Partida
        [352].S.BITS2.27   // 8-FPR-718 Cmd. Marcha
        [352].S.BITS2.20   // 8-FPR-718 Reset Falla
        [352].S.BITS2.23   // 8-FPR-718 Test
        [352].S.BITS2.30   // 8-FPR-718 OUT MARCHA
        [353].S.BITS1.2   // 8-PLT-722 Conf. Marcha
        [353].S.BITS1.29   // 110-CAN-001 Falla Abrir
        [353].S.BITS2.31   // 110-CAN-001 OUT OPEN
        [354].S.BITS1.0   // 8-BIF-724 Enable
        [354].S.BITS1.1   // 8-BIF-724 Falla Resumen
        [354].S.BITS2.20   // 8-BIF-724 Reset Falla
        [354].S.BITS2.23   // 8-BIF-724 Test
        [355].S.BITS1.2   // 110-CAN-003 Conf Pos Abrir
        [355].S.BITS1.29   // 110-CAN-003 Falla Abrir
        [355].S.BITS2.31   // 110-CAN-003 OUT OPEN
        [356].S.BITS1.2   // 8-VRT-729 Conf. Marcha
        [356].S.BITS1.29   // 110-CAN-004 Falla Abrir
        [356].S.BITS2.31   // 110-CAN-004 OUT OPEN
        [357].S.BITS1.2   // 8-ENF-730-1 Conf. Marcha
        [357].S.BITS1.29   // 110-CAN-005 Falla Abrir
        [357].S.BITS2.31   // 110-CAN-005 OUT OPEN
        [358].S.BITS1.2   // 110-CAN-006 Conf Pos Abrir
        [358].S.BITS1.29   // 110-CAN-006 Falla Abrir
        [358].S.BITS2.31   // 110-CAN-006 OUT OPEN
        [363].S.BITS1.1   // 110-CAN-008/1 Falla Resumen
        [359].S.BITS1.8   // TV LL
        [359].S.BITS1.9   // TV LM
        [359].S.BITS1.10   // TV LH
        [362].S.BITS1.8   // 110-TOL-004/1 LL
        [362].S.BITS1.9   // 110-TOL-004/1 LM
        [362].S.BITS1.10   // 110-TOL-004/1 LH
        [363].S.BITS1.0   // 110-CAN-008/1 Enable
        [363].S.BITS1.2   // 110-CAN-008/1 Conf Pos Abrir
        [363].S.BITS1.4   // 110-CAN-008/1 Conf Pos Cerrar
        [363].S.BITS1.29   // 110-CAN-008/1 Falla Abrir
        [363].S.BITS2.20   // 110-CAN-008/1 Reset Falla
        [363].S.BITS2.23   // 110-CAN-008/1 Test
        [363].S.BITS2.31   // 110-CAN-008/1 OUT OPEN
        [364].S.BITS1.0   // 8-VEN-737 Enable
        [364].S.BITS1.1   // 8-VEN-737 Falla Resumen
        [364].S.BITS1.2   // 8-VEN-737 Conf. Marcha
        [364].S.BITS1.4   // 8-VEN-737 Cmd. Automatico
        [364].S.BITS1.29   // 110-CAN-009/1 Falla Abrir
        [364].S.BITS1.30   // 8-VEN-737 Falla Partida
        [364].S.BITS2.20   // 8-VEN-737 Reset Falla
        [364].S.BITS2.23   // 8-VEN-737 Test
        [364].S.BITS2.27   // 8-VEN-737 Cmd. Marcha
        [364].S.BITS2.30   // 8-VEN-737 OUT MARCHA
        [364].S.BITS2.31   // 110-CAN-009/1 OUT OPEN
        [365].S.BITS1.0   // 8-ENF-730-2 Enable
        [365].S.BITS1.1   // 8-ENF-730-2 Falla Resumen
        [365].S.BITS1.2   // 8-ENF-730-2 Conf. Marcha
        [365].S.BITS1.4   // 8-ENF-730-2 Cmd. Automatico
        [365].S.BITS1.26   // 8-ENF-730-2 FLL
        [365].S.BITS1.27   // 8-ENF-730-2 FV0
        [365].S.BITS1.28   // 8-ENF-730-2 FATO
        [365].S.BITS1.30   // 8-ENF-730-2 Falla Partida
        [365].S.BITS2.27   // 8-ENF-730-2 Cmd. Marcha
        [365].S.BITS2.20   // 8-ENF-730-2 Reset Falla
        [365].S.BITS2.23   // 8-ENF-730-2 Test
        [365].S.BITS2.30   // 8-ENF-730-2 OUT MARCHA
        [370].S.BITS1.27   // 110-TOR-001/1 FV0
        [370].S.BITS1.0   // 110-TOR-001/1 Enable
        [370].S.BITS1.1   // 110-TOR-001/1 Falla Resumen
        [370].S.BITS1.2   // 110-TOR-001/1 Conf. Marcha
        [370].S.BITS1.4   // 110-TOR-001/1 Cmd. Automatico
        [370].S.BITS1.26   // 110-TOR-001/1 FLL
        [370].S.BITS1.28   // 110-TOR-001/1 FATO
        [370].S.BITS1.30   // 110-TOR-001/1 Falla Partida
        [370].S.BITS2.27   // 110-TOR-001/1 Cmd. Marcha
        [370].S.BITS2.20   // 110-TOR-001/1 Reset Falla
        [370].S.BITS2.23   // 110-TOR-001/1 Test
        [370].S.BITS2.30   // 110-TOR-001/1 OUT MARCHA
        [372].S.BITS1.0   // 8-VRT-746 Enable
        [372].S.BITS1.1   // 8-VRT-746 Falla Resumen
        [372].S.BITS1.2   // 8-VRT-746 Conf. Marcha
        [372].S.BITS1.4   // 8-VRT-746 Cmd. Automatico
        [372].S.BITS1.26   // 8-VRT-746 FLL
        [372].S.BITS1.27   // 8-VRT-746 FV0
        [372].S.BITS1.28   // 8-VRT-746 FATO
        [372].S.BITS1.30   // 8-VRT-746 Falla Partida
        [372].S.BITS2.27   // 8-VRT-746 Cmd. Marcha
        [372].S.BITS2.20   // 8-VRT-746 Reset Falla
        [372].S.BITS2.23   // 8-VRT-746 Test
        [372].S.BITS2.30   // 8-VRT-746 OUT MARCHA
        [373].S.BITS1.0   // 110-EXP-001/1 Enable
        [373].S.BITS1.1   // 110-EXP-001/1 Falla Resumen
        [373].S.BITS1.2   // 110-EXP-001/1 Conf. Marcha
        [373].S.BITS1.4   // 110-EXP-001/1 Cmd. Automatico
        [373].S.BITS1.26   // 110-EXP-001/1 FLL
        [373].S.BITS1.27   // 110-EXP-001/1 FV0
        [373].S.BITS1.28   // 110-EXP-001/1 FATO
        [373].S.BITS1.30   // 110-EXP-001/1 Falla Partida
        [373].S.BITS2.27   // 110-EXP-001/1 Cmd. Marcha
        [373].S.BITS2.20   // 110-EXP-001/1 Reset Falla
        [373].S.BITS2.23   // 110-EXP-001/1 Test
        [373].S.BITS2.30   // 110-EXP-001/1 OUT MARCHA
        [374].S.BITS1.0   // 8-VEN-747 Enable
        [374].S.BITS1.1   // 8-VEN-747 Falla Resumen
        [374].S.BITS1.2   // 8-VEN-747 Conf. Marcha
        [374].S.BITS1.4   // 8-VEN-747 Cmd. Automatico
        [374].S.BITS1.26   // 8-VEN-747 FLL
        [374].S.BITS1.27   // 8-VEN-747 FV0
        [374].S.BITS1.28   // 8-VEN-747 FATO
        [374].S.BITS1.30   // 8-VEN-747 Falla Partida
        [374].S.BITS2.27   // 8-VEN-747 Cmd. Marcha
        [374].S.BITS2.20   // 8-VEN-747 Reset Falla
        [374].S.BITS2.23   // 8-VEN-747 Test
        [374].S.BITS2.30   // 8-VEN-747 OUT MARCHA
        [375].S.BITS1.0   // 8-ENF-740-2 Enable
        [375].S.BITS1.1   // 8-ENF-740-2 Falla Resumen
        [375].S.BITS1.4   // 8-ENF-740-2 Cmd. Automatico
        [375].S.BITS1.26   // 8-ENF-740-2 FLL
        [375].S.BITS1.27   // 8-ENF-740-2 FV0
        [375].S.BITS1.28   // 8-ENF-740-2 FATO
        [375].S.BITS1.30   // 8-ENF-740-2 Falla Partida
        [375].S.BITS2.27   // 8-ENF-740-2 Cmd. Marcha
        [375].S.BITS2.20   // 8-ENF-740-2 Reset Falla
        [375].S.BITS2.23   // 8-ENF-740-2 Test
        [375].S.BITS2.30   // 8-ENF-740-2 OUT MARCHA
        [376].S.BITS1.0   // 8-ROS-752 Enable
        [376].S.BITS1.1   // 8-ROS-752 Falla Resumen
        [376].S.BITS1.2   // 8-ROS-752 Conf. Marcha
        [376].S.BITS1.4   // 8-ROS-752 Cmd. Automatico
        [376].S.BITS1.26   // 8-ROS-752 FLL
        [376].S.BITS1.27   // 8-ROS-752 FV0
        [376].S.BITS1.28   // 8-ROS-752 FATO
        [376].S.BITS1.30   // 8-ROS-752 Falla Partida
        [376].S.BITS2.27   // 8-ROS-752 Cmd. Marcha
        [376].S.BITS2.20   // 8-ROS-752 Reset Falla
        [376].S.BITS2.23   // 8-ROS-752 Test
        [376].S.BITS2.30   // 8-ROS-752 OUT MARCHA
        [377].S.BITS1.0   // 8-ROS-754 Enable
        [377].S.BITS1.1   // 8-ROS-754 Falla Resumen
        [377].S.BITS1.2   // 8-ROS-754 Conf. Marcha
        [377].S.BITS1.4   // 8-ROS-754 Cmd. Automatico
        [377].S.BITS1.29   // 110-BIF-001/1 Falla Pos. Izquierda
        [377].S.BITS1.30   // 8-ROS-754 Falla Partida
        [377].S.BITS2.20   // 8-ROS-754 Reset Falla
        [377].S.BITS2.23   // 8-ROS-754 Test
        [377].S.BITS2.26   // 110-BIF-001/1 Cmd. Pos . Izquierda
        [377].S.BITS2.27   // 8-ROS-754 Cmd. Marcha
        [377].S.BITS2.30   // 8-ROS-754 OUT MARCHA
        [377].S.BITS2.31   // 110-BIF-001/1 Out Derecha
        [381].S.BITS1.0   // 8-ELV-762 Enable
        [381].S.BITS1.1   // 8-ELV-762 Falla Resumen
        [381].S.BITS1.2   // 8-ELV-762 Conf. Marcha
        [381].S.BITS1.4   // 8-ELV-762 Cmd. Automatico
        [381].S.BITS1.26   // 8-ELV-762 FLL
        [381].S.BITS1.27   // 8-ELV-762 FV0
        [381].S.BITS1.28   // 8-ELV-762 FATO
        [381].S.BITS1.30   // 8-ELV-762 Falla Partida
        [381].S.BITS2.27   // 8-ELV-762 Cmd. Marcha
        [381].S.BITS2.20   // 8-ELV-762 Reset Falla
        [381].S.BITS2.23   // 8-ELV-762 Test
        [381].S.BITS2.30   // 8-ELV-762 OUT MARCHA
        [382].S.BITS1.0   // 8-ZRD-764 Enable
        [382].S.BITS1.1   // 8-ZRD-764 Falla Resumen
        [382].S.BITS1.2   // 8-ZRD-764 Conf. Marcha
        [382].S.BITS1.4   // 8-ZRD-764 Cmd. Automatico
        [382].S.BITS1.26   // 8-ZRD-764 FLL
        [382].S.BITS1.27   // 8-ZRD-764 FV0
        [382].S.BITS1.28   // 8-ZRD-764 FATO
        [382].S.BITS1.30   // 8-ZRD-764 Falla Partida
        [382].S.BITS2.27   // 8-ZRD-764 Cmd. Marcha
        [382].S.BITS2.20   // 8-ZRD-764 Reset Falla
        [382].S.BITS2.23   // 8-ZRD-764 Test
        [382].S.BITS2.30   // 8-ZRD-764 OUT MARCHA
        [384].S.BITS1.27   // 110-ENF-001/1-1 FV0
        [383].S.BITS1.8   // 110-ENF-001/1 LL
        [383].S.BITS1.9   // 110-ENF-001/1 LM
        [383].S.BITS1.10   // 110-ENF-001/1 LH
        [384].S.BITS1.0   // 8-CON-764b Enable
        [384].S.BITS1.1   // 8-CON-764b Falla Resumen
        [384].S.BITS1.2   // 8-CON-764b Conf Pos Abrir
        [384].S.BITS1.4   // 8-CON-764b Conf Pos Cerrar
        [384].S.BITS1.26   // 110-ENF-001/1-1 FLL
        [384].S.BITS1.28   // 110-ENF-001/1-1 FATO
        [384].S.BITS1.30   // 8-CON-764b Falla Cerrar
        [384].S.BITS2.27   // 8-CON-764b Cmd. Open
        [384].S.BITS2.20   // 8-CON-764b Reset Falla
        [384].S.BITS2.23   // 8-CON-764b Test
        [384].S.BITS2.30   // 8-CON-764b OUT CLOSE
        [387].S.BITS1.27   // 110-ESC-003/1 FV0
        [386].S.BITS1.8   // 110-CIC-001/1 LL
        [386].S.BITS1.9   // 110-CIC-001/1 LM
        [386].S.BITS1.10   // 110-CIC-001/1 LH
        [387].S.BITS1.0   // 9-CON-651 Enable
        [387].S.BITS1.1   // 9-CON-651 Falla Resumen
        [387].S.BITS1.2   // 9-CON-651 Conf Pos Abrir
        [387].S.BITS1.4   // 9-CON-651 Conf Pos Cerrar
        [387].S.BITS1.26   // 110-ESC-003/1 FLL
        [387].S.BITS1.28   // 110-ESC-003/1 FATO
        [387].S.BITS1.30   // 9-CON-651 Falla Cerrar
        [387].S.BITS2.27   // 9-CON-651 Cmd. Open
        [387].S.BITS2.20   // 9-CON-651 Reset Falla
        [387].S.BITS2.23   // 9-CON-651 Test
        [387].S.BITS2.30   // 9-CON-651 OUT CLOSE
        [389].S.BITS1.0   // 9-CON-653 Enable
        [389].S.BITS1.1   // 9-CON-653 Falla Resumen
        [389].S.BITS1.2   // 9-CON-653 Conf Pos Abrir
        [389].S.BITS1.4   // 9-CON-653 Conf Pos Cerrar
        [389].S.BITS1.26   // 110-VAL-001/1-1 FLL
        [389].S.BITS1.27   // 110-VAL-001/1-1 FV0
        [389].S.BITS1.28   // 110-VAL-001/1-1 FATO
        [389].S.BITS1.30   // 9-CON-653 Falla Cerrar
        [389].S.BITS2.27   // 9-CON-653 Cmd. Open
        [389].S.BITS2.20   // 9-CON-653 Reset Falla
        [389].S.BITS2.23   // 9-CON-653 Test
        [389].S.BITS2.30   // 9-CON-653 OUT CLOSE
        [390].S.BITS1.0   // 9-CON-654 Enable
        [390].S.BITS1.1   // 9-CON-654 Falla Resumen
        [390].S.BITS1.2   // 9-CON-654 Conf Pos Abrir
        [390].S.BITS1.4   // 9-CON-654 Conf Pos Cerrar
        [390].S.BITS1.26   // 110-VEN-001/1-1 FLL
        [390].S.BITS1.27   // 110-VEN-001/1-1 FV0
        [390].S.BITS1.28   // 110-VEN-001/1-1 FATO
        [390].S.BITS1.30   // 9-CON-654 Falla Cerrar
        [390].S.BITS2.27   // 9-CON-654 Cmd. Open
        [390].S.BITS2.20   // 9-CON-654 Reset Falla
        [390].S.BITS2.23   // 9-CON-654 Test
        [390].S.BITS2.30   // 9-CON-654 OUT CLOSE
        [391].S.BITS1.0   // 110-ENF-001/1-5 Enable
        [391].S.BITS1.1   // 110-ENF-001/1-5 Falla Resumen
        [391].S.BITS1.2   // 110-ENF-001/1-5 Conf. Marcha
        [391].S.BITS1.4   // 110-ENF-001/1-5 Cmd. Automatico
        [391].S.BITS1.26   // 110-ENF-001/1-5 FLL
        [391].S.BITS1.27   // 110-ENF-001/1-5 FV0
        [391].S.BITS1.28   // 110-ENF-001/1-5 FATO
        [391].S.BITS1.30   // 110-ENF-001/1-5 Falla Partida
        [391].S.BITS2.27   // 110-ENF-001/1-5 Cmd. Marcha
        [391].S.BITS2.20   // 110-ENF-001/1-5 Reset Falla
        [391].S.BITS2.23   // 110-ENF-001/1-5 Test
        [391].S.BITS2.30   // 110-ENF-001/1-5 OUT MARCHA
        [401].S.BITS1.0   // 9-CON-663 Enable
        [401].S.BITS1.1   // 9-CON-663 Falla Resumen
        [401].S.BITS1.2   // 9-CON-663 Conf Pos Abrir
        [401].S.BITS1.4   // 9-CON-663 Conf Pos Cerrar
        [401].S.BITS1.26   // 110-ESC-002/1 FLL
        [401].S.BITS1.27   // 110-ESC-002/1 FV0
        [401].S.BITS1.28   // 110-ESC-002/1 FATO
        [401].S.BITS1.30   // 9-CON-663 Falla Cerrar
        [401].S.BITS2.27   // 9-CON-663 Cmd. Open
        [401].S.BITS2.20   // 9-CON-663 Reset Falla
        [401].S.BITS2.23   // 9-CON-663 Test
        [401].S.BITS2.30   // 9-CON-663 OUT CLOSE
        [402].S.BITS1.0   // 9-CON-664 Enable
        [402].S.BITS1.1   // 9-CON-664 Falla Resumen
        [402].S.BITS1.2   // 9-CON-664 Conf Pos Abrir
        [402].S.BITS1.4   // 9-CON-664 Conf Pos Cerrar
        [402].S.BITS1.26   // 110-ENF-002/1-4 FLL
        [402].S.BITS1.27   // 110-ENF-002/1-4 FV0
        [402].S.BITS1.28   // 110-ENF-002/1-4 FATO
        [402].S.BITS1.30   // 9-CON-664 Falla Cerrar
        [402].S.BITS2.27   // 9-CON-664 Cmd. Open
        [402].S.BITS2.20   // 9-CON-664 Reset Falla
        [402].S.BITS2.23   // 9-CON-664 Test
        [402].S.BITS2.30   // 9-CON-664 OUT CLOSE
        [404].S.BITS1.27   // 110-ENF-002/1-1 FV0
        [403].S.BITS1.8   // 110-ENF-002/1 LL
        [403].S.BITS1.9   // 110-ENF-002/1 LM
        [403].S.BITS1.10   // 110-ENF-002/1 LH
        [404].S.BITS1.0   // 9-CON-666 Enable
        [404].S.BITS1.1   // 9-CON-666 Falla Resumen
        [404].S.BITS1.2   // 9-CON-666 Conf Pos Abrir
        [404].S.BITS1.4   // 9-CON-666 Conf Pos Cerrar
        [404].S.BITS1.26   // 110-ENF-002/1-1 FLL
        [404].S.BITS1.28   // 110-ENF-002/1-1 FATO
        [404].S.BITS1.30   // 9-CON-666 Falla Cerrar
        [404].S.BITS2.27   // 9-CON-666 Cmd. Open
        [404].S.BITS2.20   // 9-CON-666 Reset Falla
        [404].S.BITS2.23   // 9-CON-666 Test
        [404].S.BITS2.30   // 9-CON-666 OUT CLOSE
        [407].S.BITS1.27   // 110-ESC-004/1 FV0
        [406].S.BITS1.8   // 110-CIC-002/1 LL
        [406].S.BITS1.9   // 110-CIC-002/1 LM
        [406].S.BITS1.10   // 110-CIC-002/1 LH
        [407].S.BITS1.0   // 110-ESC-004/1 Enable
        [407].S.BITS1.1   // 110-ESC-004/1 Falla Resumen
        [407].S.BITS1.2   // 110-ESC-004/1 Conf. Marcha
        [407].S.BITS1.4   // 110-ESC-004/1 Cmd. Automatico
        [407].S.BITS1.26   // 110-ESC-004/1 FLL
        [407].S.BITS1.28   // 110-ESC-004/1 FATO
        [407].S.BITS1.30   // 110-ESC-004/1 Falla Partida
        [407].S.BITS2.27   // 110-ESC-004/1 Cmd. Marcha
        [407].S.BITS2.20   // 110-ESC-004/1 Reset Falla
        [407].S.BITS2.23   // 110-ESC-004/1 Test
        [407].S.BITS2.30   // 110-ESC-004/1 OUT MARCHA
        [409].S.BITS1.0   // 9-CON-671 Enable
        [409].S.BITS1.1   // 9-CON-671 Falla Resumen
        [409].S.BITS1.2   // 9-CON-671 Conf Pos Abrir
        [409].S.BITS1.4   // 9-CON-671 Conf Pos Cerrar
        [409].S.BITS1.26   // 110-VAL-002/1-1 FLL
        [409].S.BITS1.27   // 110-VAL-002/1-1 FV0
        [409].S.BITS1.28   // 110-VAL-002/1-1 FATO
        [409].S.BITS1.30   // 9-CON-671 Falla Cerrar
        [409].S.BITS2.27   // 9-CON-671 Cmd. Open
        [409].S.BITS2.20   // 9-CON-671 Reset Falla
        [409].S.BITS2.23   // 9-CON-671 Test
        [409].S.BITS2.30   // 9-CON-671 OUT CLOSE
        [410].S.BITS1.0   // 9-CON-672 Enable
        [410].S.BITS1.1   // 9-CON-672 Falla Resumen
        [410].S.BITS1.2   // 9-CON-672 Conf Pos Abrir
        [410].S.BITS1.4   // 9-CON-672 Conf Pos Cerrar
        [410].S.BITS1.26   // 110-VEN-002/1-1 FLL
        [410].S.BITS1.27   // 110-VEN-002/1-1 FV0
        [410].S.BITS1.28   // 110-VEN-002/1-1 FATO
        [410].S.BITS1.30   // 9-CON-672 Falla Cerrar
        [410].S.BITS2.27   // 9-CON-672 Cmd. Open
        [410].S.BITS2.20   // 9-CON-672 Reset Falla
        [410].S.BITS2.23   // 9-CON-672 Test
        [410].S.BITS2.30   // 9-CON-672 OUT CLOSE
        [411].S.BITS1.0   // 9-CON-673 Enable
        [411].S.BITS1.1   // 9-CON-673 Falla Resumen
        [411].S.BITS1.2   // 9-CON-673 Conf Pos Abrir
        [411].S.BITS1.4   // 9-CON-673 Conf Pos Cerrar
        [411].S.BITS1.26   // 110-ENF-002/1-5 FLL
        [411].S.BITS1.27   // 110-ENF-002/1-5 FV0
        [411].S.BITS1.28   // 110-ENF-002/1-5 FATO
        [411].S.BITS1.30   // 9-CON-673 Falla Cerrar
        [411].S.BITS2.27   // 9-CON-673 Cmd. Open
        [411].S.BITS2.20   // 9-CON-673 Reset Falla
        [411].S.BITS2.23   // 9-CON-673 Test
        [411].S.BITS2.30   // 9-CON-673 OUT CLOSE
        [414].S.BITS1.0   // 9-CON-676 Enable
        [414].S.BITS1.1   // 9-CON-676 Falla Resumen
        [414].S.BITS1.2   // 9-CON-676 Conf Pos Abrir
        [414].S.BITS1.4   // 9-CON-676 Conf Pos Cerrar
        [414].S.BITS1.26   // 110-TOR-002/1 FLL
        [414].S.BITS1.27   // 110-TOR-002/1 FV0
        [414].S.BITS1.28   // 110-TOR-002/1 FATO
        [414].S.BITS1.30   // 9-CON-676 Falla Cerrar
        [414].S.BITS2.27   // 9-CON-676 Cmd. Open
        [414].S.BITS2.20   // 9-CON-676 Reset Falla
        [414].S.BITS2.23   // 9-CON-676 Test
        [414].S.BITS2.30   // 9-CON-676 OUT CLOSE
        [415].S.BITS1.0   // 9-CON-677 Enable
        [415].S.BITS1.1   // 9-CON-677 Falla Resumen
        [415].S.BITS1.2   // 9-CON-677 Conf Pos Abrir
        [415].S.BITS1.4   // 9-CON-677 Conf Pos Cerrar
        [415].S.BITS1.26   // 110-TOR-003/1 FLL
        [415].S.BITS1.27   // 110-TOR-003/1 FV0
        [415].S.BITS1.28   // 110-TOR-003/1 FATO
        [415].S.BITS1.30   // 9-CON-677 Falla Cerrar
        [415].S.BITS2.27   // 9-CON-677 Cmd. Open
        [415].S.BITS2.20   // 9-CON-677 Reset Falla
        [415].S.BITS2.23   // 9-CON-677 Test
        [415].S.BITS2.30   // 9-CON-677 OUT CLOSE
        [416].S.BITS1.0   // 9-CON-678 Enable
        [416].S.BITS1.1   // 9-CON-678 Falla Resumen
        [416].S.BITS1.2   // 9-CON-678 Conf Pos Abrir
        [416].S.BITS1.4   // 9-CON-678 Conf Pos Cerrar
        [416].S.BITS1.26   // 110-ELV-002/1 FLL
        [416].S.BITS1.27   // 110-ELV-002/1 FV0
        [416].S.BITS1.28   // 110-ELV-002/1 FATO
        [416].S.BITS1.30   // 9-CON-678 Falla Cerrar
        [416].S.BITS2.27   // 9-CON-678 Cmd. Open
        [416].S.BITS2.20   // 9-CON-678 Reset Falla
        [416].S.BITS2.23   // 9-CON-678 Test
        [416].S.BITS2.30   // 9-CON-678 OUT CLOSE
        [417].S.BITS1.0   // 110-TOL-006/1 Enable
        [417].S.BITS1.1   // 110-TOL-006/1 Falla Resumen
        [417].S.BITS1.2   // 110-TOL-006/1 Conf. Marcha
        [417].S.BITS1.4   // 110-TOL-006/1 Cmd. Automatico
        [417].S.BITS1.26   // 110-TOL-006/1 FLL
        [417].S.BITS1.27   // 110-TOL-006/1 FV0
        [417].S.BITS1.28   // 110-TOL-006/1 FATO
        [417].S.BITS1.30   // 110-TOL-006/1 Falla Partida
        [417].S.BITS2.27   // 110-TOL-006/1 Cmd. Marcha
        [417].S.BITS2.20   // 110-TOL-006/1 Reset Falla
        [417].S.BITS2.23   // 110-TOL-006/1 Test
        [417].S.BITS2.30   // 110-TOL-006/1 OUT MARCHA
        [418].S.BITS1.0   // 9-RED-680 Enable
        [418].S.BITS1.1   // 9-RED-680 Falla Resumen
        [418].S.BITS1.2   // 9-RED-680 Conf. Marcha
        [418].S.BITS1.4   // 9-RED-680 Cmd. Automatico
        [418].S.BITS1.26   // 9-RED-680 FLL
        [418].S.BITS1.27   // 9-RED-680 FV0
        [418].S.BITS1.28   // 9-RED-680 FATO
        [418].S.BITS1.30   // 9-RED-680 Falla Partida
        [418].S.BITS2.27   // 9-RED-680 Cmd. Marcha
        [418].S.BITS2.20   // 9-RED-680 Reset Falla
        [418].S.BITS2.23   // 9-RED-680 Test
        [418].S.BITS2.30   // 9-RED-680 OUT MARCHA
        [423].S.BITS1.30   // 9-CON-685 Falla Cerrar
        [422].S.BITS1.8   // 110-TOL-004/2 LL
        [422].S.BITS1.9   // 110-TOL-004/2 LM
        [422].S.BITS1.10   // 110-TOL-004/2 LH
        [423].S.BITS1.0   // 9-CON-685 Enable
        [423].S.BITS1.1   // 9-CON-685 Falla Resumen
        [423].S.BITS1.2   // 9-CON-685 Conf Pos Abrir
        [423].S.BITS1.4   // 9-CON-685 Conf Pos Cerrar
        [423].S.BITS1.29   // 9-CON-685 Falla Abrir
        [423].S.BITS2.20   // 9-CON-685 Reset Falla
        [423].S.BITS2.23   // 9-CON-685 Test
        [423].S.BITS2.27   // 9-CON-685 Cmd. Open
        [423].S.BITS2.30   // 9-CON-685 OUT CLOSE
        [423].S.BITS2.31   // 9-CON-685 OUT OPEN
        [424].S.BITS1.0   // 9-CON-686 Enable
        [424].S.BITS1.1   // 9-CON-686 Falla Resumen
        [424].S.BITS1.2   // 9-CON-686 Conf Pos Abrir
        [424].S.BITS1.4   // 9-CON-686 Conf Pos Cerrar
        [424].S.BITS1.29   // 9-CON-686 Falla Abrir
        [424].S.BITS1.30   // 9-CON-686 Falla Cerrar
        [424].S.BITS2.20   // 9-CON-686 Reset Falla
        [424].S.BITS2.23   // 9-CON-686 Test
        [424].S.BITS2.27   // 9-CON-686 Cmd. Open
        [424].S.BITS2.30   // 9-CON-686 OUT CLOSE
        [424].S.BITS2.31   // 9-CON-686 OUT OPEN
        [425].S.BITS1.0   // 9-CON-687 Enable
        [425].S.BITS1.1   // 9-CON-687 Falla Resumen
        [425].S.BITS1.2   // 9-CON-687 Conf Pos Abrir
        [425].S.BITS1.4   // 9-CON-687 Conf Pos Cerrar
        [425].S.BITS1.26   // 110-CAN-010/2 FLL
        [425].S.BITS1.27   // 110-CAN-010/2 FV0
        [425].S.BITS1.28   // 110-CAN-010/2 FATO
        [425].S.BITS1.30   // 9-CON-687 Falla Cerrar
        [425].S.BITS2.27   // 9-CON-687 Cmd. Open
        [425].S.BITS2.20   // 9-CON-687 Reset Falla
        [425].S.BITS2.23   // 9-CON-687 Test
        [425].S.BITS2.30   // 9-CON-687 OUT CLOSE
        [430].S.BITS1.27   // 110-TOR-001/2 FV0
        [429].S.BITS1.8   // 110-TOL-005/2 LL
        [429].S.BITS1.9   // 110-TOL-005/2 LM
        [429].S.BITS1.10   // 110-TOL-005/2 LH
        [430].S.BITS1.0   // 9-CON-692 Enable
        [430].S.BITS1.1   // 9-CON-692 Falla Resumen
        [430].S.BITS1.2   // 9-CON-692 Conf Pos Abrir
        [430].S.BITS1.4   // 9-CON-692 Conf Pos Cerrar
        [430].S.BITS1.26   // 110-TOR-001/2 FLL
        [430].S.BITS1.28   // 110-TOR-001/2 FATO
        [430].S.BITS1.30   // 9-CON-692 Falla Cerrar
        [430].S.BITS2.27   // 9-CON-692 Cmd. Open
        [430].S.BITS2.20   // 9-CON-692 Reset Falla
        [430].S.BITS2.23   // 9-CON-692 Test
        [430].S.BITS2.30   // 9-CON-692 OUT CLOSE
        [432].S.BITS1.0   // 9-CON-694 Enable
        [432].S.BITS1.1   // 9-CON-694 Falla Resumen
        [432].S.BITS1.2   // 9-CON-694 Conf Pos Abrir
        [432].S.BITS1.4   // 9-CON-694 Conf Pos Cerrar
        [432].S.BITS1.26   // 110-ACD-001/2 FLL
        [432].S.BITS1.27   // 110-ACD-001/2 FV0
        [432].S.BITS1.28   // 110-ACD-001/2 FATO
        [432].S.BITS1.30   // 9-CON-694 Falla Cerrar
        [432].S.BITS2.27   // 9-CON-694 Cmd. Open
        [432].S.BITS2.20   // 9-CON-694 Reset Falla
        [432].S.BITS2.23   // 9-CON-694 Test
        [432].S.BITS2.30   // 9-CON-694 OUT CLOSE
        [433].S.BITS1.0   // 9-CON-695 Enable
        [433].S.BITS1.1   // 9-CON-695 Falla Resumen
        [433].S.BITS1.2   // 9-CON-695 Conf Pos Abrir
        [433].S.BITS1.4   // 9-CON-695 Conf Pos Cerrar
        [433].S.BITS1.26   // 110-EXP-001/2 FLL
        [433].S.BITS1.27   // 110-EXP-001/2 FV0
        [433].S.BITS1.28   // 110-EXP-001/2 FATO
        [433].S.BITS1.30   // 9-CON-695 Falla Cerrar
        [433].S.BITS2.27   // 9-CON-695 Cmd. Open
        [433].S.BITS2.20   // 9-CON-695 Reset Falla
        [433].S.BITS2.23   // 9-CON-695 Test
        [433].S.BITS2.30   // 9-CON-695 OUT CLOSE
        [434].S.BITS1.0   // 9-CON-696 Enable
        [434].S.BITS1.1   // 9-CON-696 Falla Resumen
        [434].S.BITS1.2   // 9-CON-696 Conf Pos Abrir
        [434].S.BITS1.4   // 9-CON-696 Conf Pos Cerrar
        [434].S.BITS1.26   // 110-DES-001/2 FLL
        [434].S.BITS1.27   // 110-DES-001/2 FV0
        [434].S.BITS1.28   // 110-DES-001/2 FATO
        [434].S.BITS1.30   // 9-CON-696 Falla Cerrar
        [434].S.BITS2.27   // 9-CON-696 Cmd. Open
        [434].S.BITS2.20   // 9-CON-696 Reset Falla
        [434].S.BITS2.23   // 9-CON-696 Test
        [434].S.BITS2.30   // 9-CON-696 OUT CLOSE
        [435].S.BITS1.0   // 9-CON-697 Enable
        [435].S.BITS1.1   // 9-CON-697 Falla Resumen
        [435].S.BITS1.2   // 9-CON-697 Conf Pos Abrir
        [435].S.BITS1.4   // 9-CON-697 Conf Pos Cerrar
        [435].S.BITS1.26   // 110-CAE-001/2 FLL
        [435].S.BITS1.27   // 110-CAE-001/2 FV0
        [435].S.BITS1.28   // 110-CAE-001/2 FATO
        [435].S.BITS1.30   // 9-CON-697 Falla Cerrar
        [435].S.BITS2.27   // 9-CON-697 Cmd. Open
        [435].S.BITS2.20   // 9-CON-697 Reset Falla
        [435].S.BITS2.23   // 9-CON-697 Test
        [435].S.BITS2.30   // 9-CON-697 OUT CLOSE
        [436].S.BITS1.0   // 9-CON-698 Enable
        [436].S.BITS1.1   // 9-CON-698 Falla Resumen
        [436].S.BITS1.2   // 9-CON-698 Conf Pos Abrir
        [436].S.BITS1.4   // 9-CON-698 Conf Pos Cerrar
        [436].S.BITS1.26   // 110-PLT-001/2 FLL
        [436].S.BITS1.27   // 110-PLT-001/2 FV0
        [436].S.BITS1.28   // 110-PLT-001/2 FATO
        [436].S.BITS1.30   // 9-CON-698 Falla Cerrar
        [436].S.BITS2.27   // 9-CON-698 Cmd. Open
        [436].S.BITS2.20   // 9-CON-698 Reset Falla
        [436].S.BITS2.23   // 9-CON-698 Test
        [436].S.BITS2.30   // 9-CON-698 OUT CLOSE
        [437].S.BITS1.0   // 110-BIF-001/2 Enable
        [437].S.BITS1.1   // 110-BIF-001/2 Falla Resumen
        [437].S.BITS1.2   // 110-BIF-001/2 Conf. Pos. Izquierda
        [437].S.BITS1.4   // 110-BIF-001/2 Conf. Pos. Derecha
        [437].S.BITS1.29   // 110-BIF-001/2 Falla Pos. Izquierda
        [437].S.BITS1.30   // 110-BIF-001/2 Falla Pos. Derecha
        [437].S.BITS2.20   // 110-BIF-001/2 Reset Falla
        [437].S.BITS2.23   // 110-BIF-001/2 Test
        [437].S.BITS2.26   // 110-BIF-001/2 Cmd. Pos . Izquierda
        [437].S.BITS2.27   // 110-BIF-001/2 Cmd. Pos. Derecha
        [437].S.BITS2.30   // 110-BIF-001/2 Out Izquierda
        [437].S.BITS2.31   // 110-BIF-001/2 Out Derecha
        [441].S.BITS1.0   // 9-CON-703 Enable
        [441].S.BITS1.1   // 9-CON-703 Falla Resumen
        [441].S.BITS1.2   // 9-CON-703 Conf Pos Abrir
        [441].S.BITS1.4   // 9-CON-703 Conf Pos Cerrar
        [441].S.BITS1.26   // 110-ESC-001/2 FLL
        [441].S.BITS1.27   // 110-ESC-001/2 FV0
        [441].S.BITS1.28   // 110-ESC-001/2 FATO
        [441].S.BITS1.30   // 9-CON-703 Falla Cerrar
        [441].S.BITS2.27   // 9-CON-703 Cmd. Open
        [441].S.BITS2.20   // 9-CON-703 Reset Falla
        [441].S.BITS2.23   // 9-CON-703 Test
        [441].S.BITS2.30   // 9-CON-703 OUT CLOSE
        [442].S.BITS1.0   // 110-ENF-001/2-4 Enable
        [442].S.BITS1.1   // 110-ENF-001/2-4 Falla Resumen
        [442].S.BITS1.2   // 110-ENF-001/2-4 Conf. Marcha
        [442].S.BITS1.4   // 110-ENF-001/2-4 Cmd. Automatico
        [442].S.BITS1.26   // 110-ENF-001/2-4 FLL
        [442].S.BITS1.27   // 110-ENF-001/2-4 FV0
        [442].S.BITS1.28   // 110-ENF-001/2-4 FATO
        [442].S.BITS1.30   // 110-ENF-001/2-4 Falla Partida
        [442].S.BITS2.27   // 110-ENF-001/2-4 Cmd. Marcha
        [442].S.BITS2.20   // 110-ENF-001/2-4 Reset Falla
        [442].S.BITS2.23   // 110-ENF-001/2-4 Test
        [442].S.BITS2.30   // 110-ENF-001/2-4 OUT MARCHA
        [444].S.BITS1.27   // 110-ENF-001/2-1 FV0
        [443].S.BITS1.8   // 110-ENF-001/2 LL
        [443].S.BITS1.9   // 110-ENF-001/2 LM
